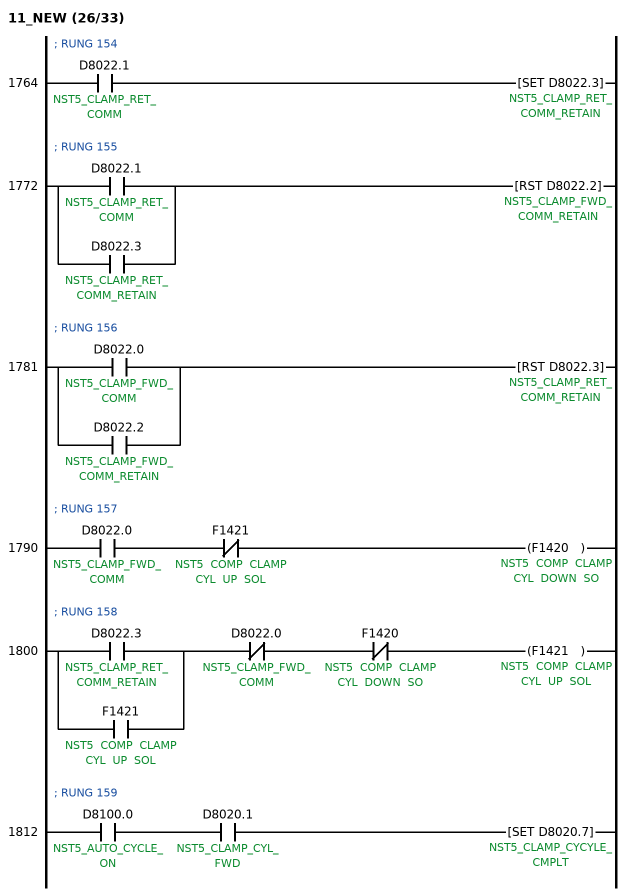
[picture p216: ladder of 11_NEW, rungs at steps 1764 to 1812]
; RUNG 154
1764  LD      D8022.1  ; NST5_CLAMP_RET_COMM
      SET     D8022.3  ; NST5_CLAMP_RET_COMM_RETAIN
; RUNG 155
1772  LD      D8022.1  ; NST5_CLAMP_RET_COMM
      OR      D8022.3  ; NST5_CLAMP_RET_COMM_RETAIN
      RST     D8022.2  ; NST5_CLAMP_FWD_COMM_RETAIN
; RUNG 156
1781  LD      D8022.0  ; NST5_CLAMP_FWD_COMM
      OR      D8022.2  ; NST5_CLAMP_FWD_COMM_RETAIN
      RST     D8022.3  ; NST5_CLAMP_RET_COMM_RETAIN
; RUNG 157
1790  LD      D8022.0  ; NST5_CLAMP_FWD_COMM
      ANI     F1421  ; NST5  COMP  CLAMP  CYL  UP  SOL
      OUT     F1420  ; NST5  COMP  CLAMP  CYL  DOWN  SO
; RUNG 158
1800  LD      D8022.3  ; NST5_CLAMP_RET_COMM_RETAIN
      OR      F1421  ; NST5  COMP  CLAMP  CYL  UP  SOL
      ANI     D8022.0  ; NST5_CLAMP_FWD_COMM
      ANI     F1420  ; NST5  COMP  CLAMP  CYL  DOWN  SO
      OUT     F1421  ; NST5  COMP  CLAMP  CYL  UP  SOL
; RUNG 159
1812  LD      D8100.0  ; NST5_AUTO_CYCLE_ON
      AND     D8020.1  ; NST5_CLAMP_CYL_FWD
      SET     D8020.7  ; NST5_CLAMP_CYCYLE_CMPLT
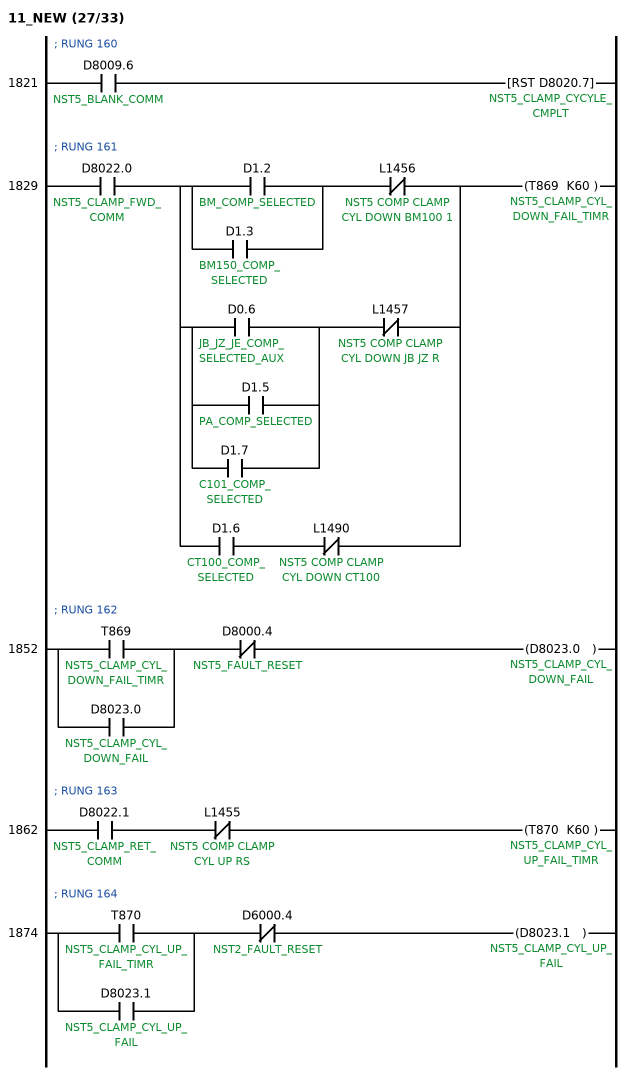
; RUNG 160
1821  LD      D8009.6  ; NST5_BLANK_COMM
      RST     D8020.7  ; NST5_CLAMP_CYCYLE_CMPLT
; RUNG 161
1829  LD      D8022.0  ; NST5_CLAMP_FWD_COMM
      LD      D1.2  ; BM_COMP_SELECTED
      OR      D1.3  ; BM150_COMP_SELECTED
      ANI     L1456  ; NST5 COMP CLAMP CYL DOWN BM100 1
      LD      D0.6  ; JB_JZ_JE_COMP_SELECTED_AUX
      OR      D1.5  ; PA_COMP_SELECTED
      OR      D1.7  ; C101_COMP_SELECTED
      ANI     L1457  ; NST5 COMP CLAMP CYL DOWN JB JZ R
      ORB
      LD      D1.6  ; CT100_COMP_SELECTED
      ANI     L1490  ; NST5 COMP CLAMP CYL DOWN CT100
      ORB
      ANB
      OUT     T869 K60  ; NST5_CLAMP_CYL_DOWN_FAIL_TIMR
; RUNG 162
1852  LD      T869  ; NST5_CLAMP_CYL_DOWN_FAIL_TIMR
      OR      D8023.0  ; NST5_CLAMP_CYL_DOWN_FAIL
      ANI     D8000.4  ; NST5_FAULT_RESET
      OUT     D8023.0  ; NST5_CLAMP_CYL_DOWN_FAIL
; RUNG 163
1862  LD      D8022.1  ; NST5_CLAMP_RET_COMM
      ANI     L1455  ; NST5 COMP CLAMP CYL UP RS
      OUT     T870 K60  ; NST5_CLAMP_CYL_UP_FAIL_TIMR
; RUNG 164
1874  LD      T870  ; NST5_CLAMP_CYL_UP_FAIL_TIMR
      OR      D8023.1  ; NST5_CLAMP_CYL_UP_FAIL
      ANI     D6000.4  ; NST2_FAULT_RESET
      OUT     D8023.1  ; NST5_CLAMP_CYL_UP_FAIL
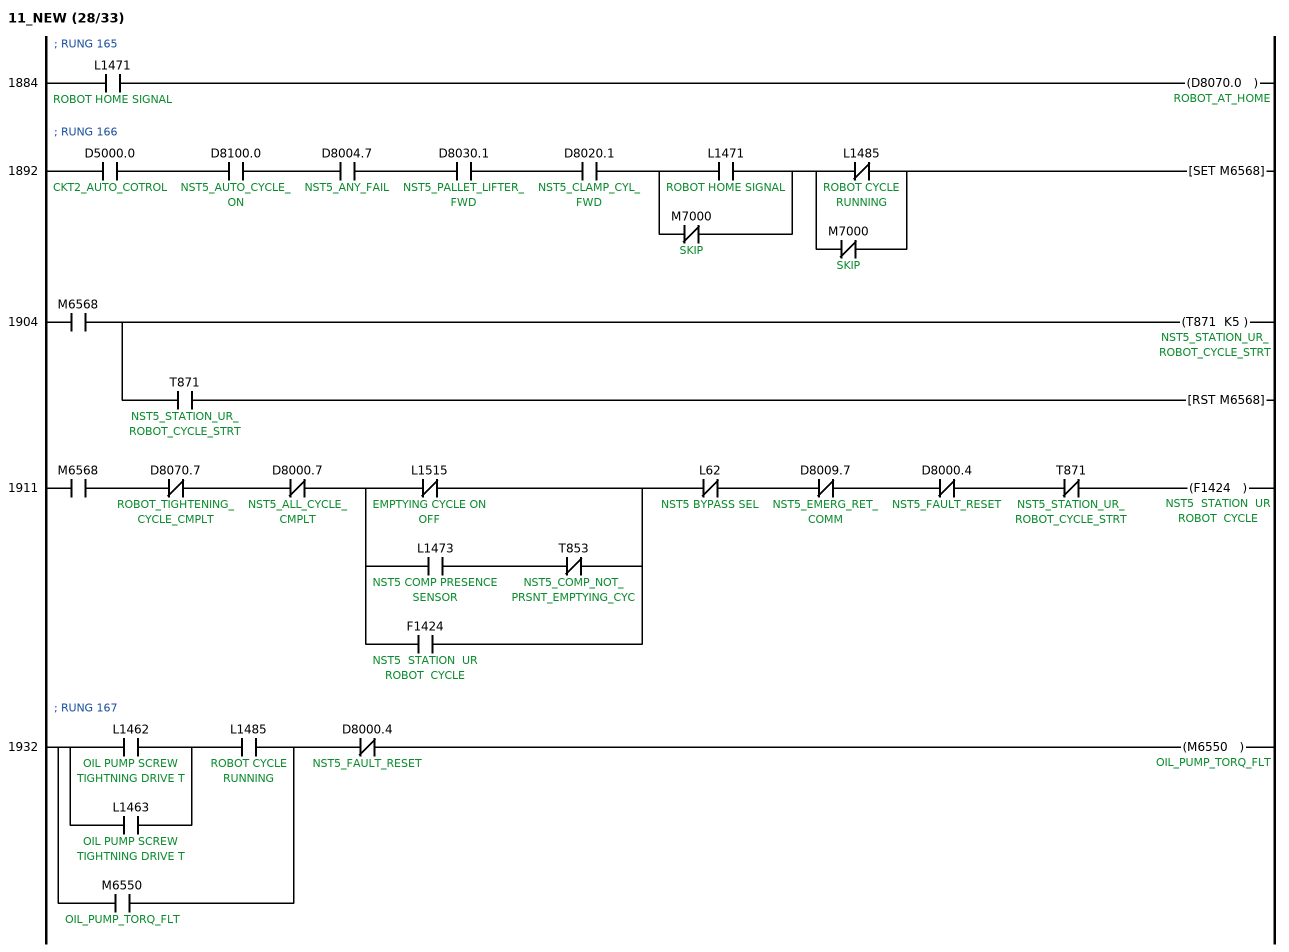
; RUNG 165
1884  LD      L1471  ; ROBOT HOME SIGNAL
      OUT     D8070.0  ; ROBOT_AT_HOME
; RUNG 166
1892  LD      D5000.0  ; CKT2_AUTO_COTROL
      AND     D8100.0  ; NST5_AUTO_CYCLE_ON
      AND     D8004.7  ; NST5_ANY_FAIL
      AND     D8030.1  ; NST5_PALLET_LIFTER_FWD
      AND     D8020.1  ; NST5_CLAMP_CYL_FWD
      LD      L1471  ; ROBOT HOME SIGNAL
      ORI     M7000  ; SKIP
      ANB
      LDI     L1485  ; ROBOT CYCLE RUNNING
      ORI     M7000  ; SKIP
      ANB
      SET     M6568
1904  LD      M6568
      OUT     T871 K5  ; NST5_STATION_UR_ROBOT_CYCLE_STRT
      AND     T871  ; NST5_STATION_UR_ROBOT_CYCLE_STRT
      RST     M6568
1911  LD      M6568
      ANI     D8070.7  ; ROBOT_TIGHTENING_CYCLE_CMPLT
      ANI     D8000.7  ; NST5_ALL_CYCLE_CMPLT
      LDI     L1515  ; EMPTYING CYCLE ON OFF
      LD      L1473  ; NST5 COMP PRESENCE SENSOR
      ANI     T853  ; NST5_COMP_NOT_PRSNT_EMPTYING_CYC
      ORB
      OR      F1424  ; NST5  STATION  UR  ROBOT  CYCLE
      ANB
      ANI     L62  ; NST5 BYPASS SEL
      ANI     D8009.7  ; NST5_EMERG_RET_COMM
      ANI     D8000.4  ; NST5_FAULT_RESET
      ANI     T871  ; NST5_STATION_UR_ROBOT_CYCLE_STRT
      OUT     F1424  ; NST5  STATION  UR  ROBOT  CYCLE
; RUNG 167
1932  LD      L1462  ; OIL PUMP SCREW TIGHTNING DRIVE T
      OR      L1463  ; OIL PUMP SCREW TIGHTNING DRIVE T
      AND     L1485  ; ROBOT CYCLE RUNNING
      OR      M6550  ; OIL_PUMP_TORQ_FLT
      ANI     D8000.4  ; NST5_FAULT_RESET
      OUT     M6550  ; OIL_PUMP_TORQ_FLT
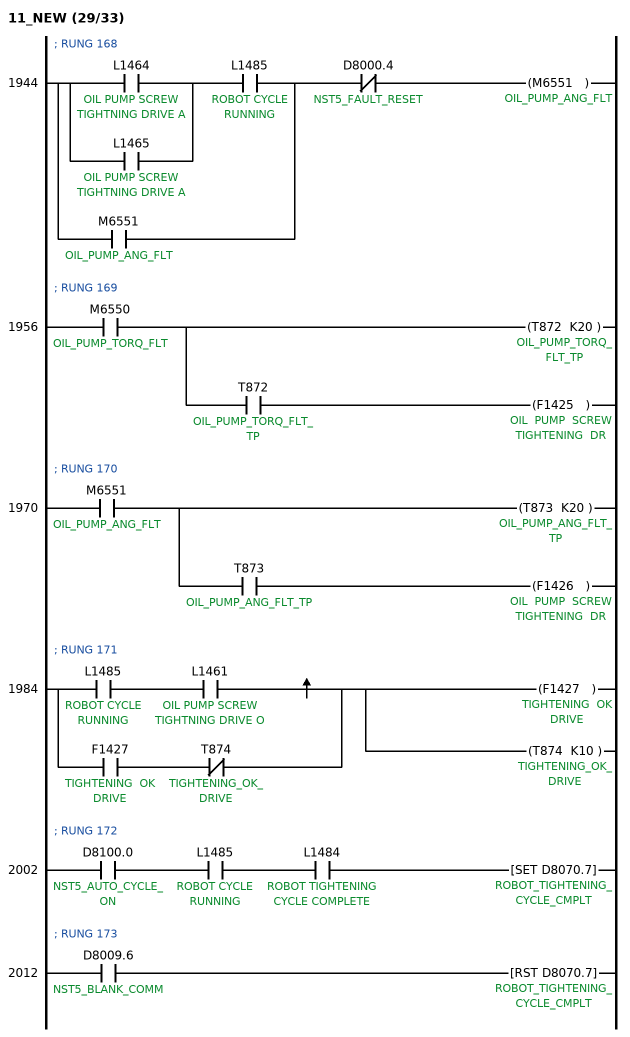
; RUNG 168
1944  LD      L1464  ; OIL PUMP SCREW TIGHTNING DRIVE A
      OR      L1465  ; OIL PUMP SCREW TIGHTNING DRIVE A
      AND     L1485  ; ROBOT CYCLE RUNNING
      OR      M6551  ; OIL_PUMP_ANG_FLT
      ANI     D8000.4  ; NST5_FAULT_RESET
      OUT     M6551  ; OIL_PUMP_ANG_FLT
; RUNG 169
1956  LD      M6550  ; OIL_PUMP_TORQ_FLT
      OUT     T872 K20  ; OIL_PUMP_TORQ_FLT_TP
      AND     T872  ; OIL_PUMP_TORQ_FLT_TP
      OUT     F1425  ; OIL  PUMP  SCREW  TIGHTENING  DR
; RUNG 170
1970  LD      M6551  ; OIL_PUMP_ANG_FLT
      OUT     T873 K20  ; OIL_PUMP_ANG_FLT_TP
      AND     T873  ; OIL_PUMP_ANG_FLT_TP
      OUT     F1426  ; OIL  PUMP  SCREW  TIGHTENING  DR
; RUNG 171
1984  LD      L1485  ; ROBOT CYCLE RUNNING
      AND     L1461  ; OIL PUMP SCREW TIGHTNING DRIVE O
      MEP
      LD      F1427  ; TIGHTENING  OK  DRIVE
      ANI     T874  ; TIGHTENING_OK_DRIVE
      ORB
      OUT     F1427  ; TIGHTENING  OK  DRIVE
      OUT     T874 K10  ; TIGHTENING_OK_DRIVE
; RUNG 172
2002  LD      D8100.0  ; NST5_AUTO_CYCLE_ON
      AND     L1485  ; ROBOT CYCLE RUNNING
      AND     L1484  ; ROBOT TIGHTENING CYCLE COMPLETE
      SET     D8070.7  ; ROBOT_TIGHTENING_CYCLE_CMPLT
; RUNG 173
2012  LD      D8009.6  ; NST5_BLANK_COMM
      RST     D8070.7  ; ROBOT_TIGHTENING_CYCLE_CMPLT
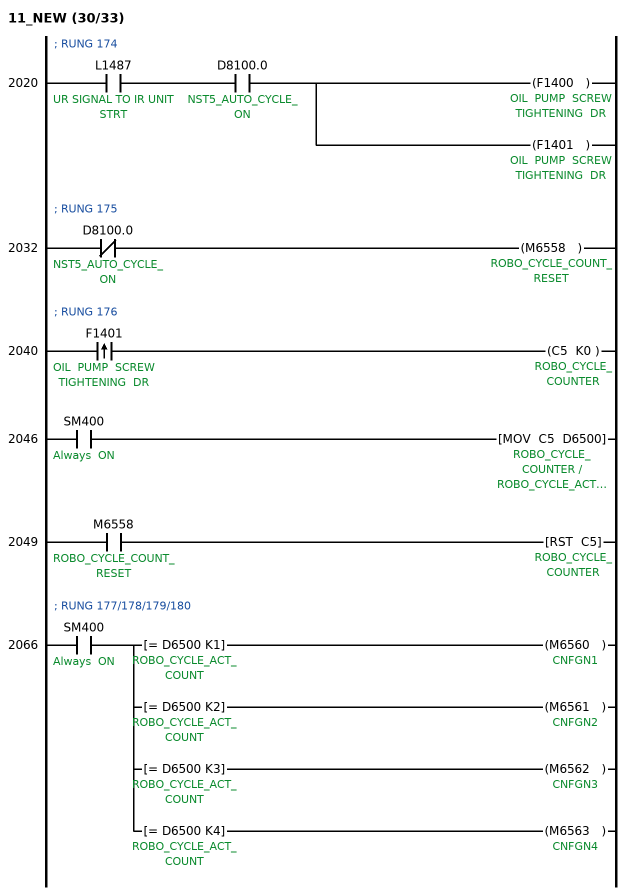
; RUNG 174
2020  LD      L1487  ; UR SIGNAL TO IR UNIT STRT
      AND     D8100.0  ; NST5_AUTO_CYCLE_ON
      OUT     F1400  ; OIL  PUMP  SCREW  TIGHTENING  DR
      OUT     F1401  ; OIL  PUMP  SCREW  TIGHTENING  DR
; RUNG 175
2032  LDI     D8100.0  ; NST5_AUTO_CYCLE_ON
      OUT     M6558  ; ROBO_CYCLE_COUNT_RESET
; RUNG 176
2040  LDP     F1401  ; OIL  PUMP  SCREW  TIGHTENING  DR
      OUT     C5 K0  ; ROBO_CYCLE_COUNTER
2046  LD      SM400  ; Always  ON
      MOV     C5 D6500  ; ROBO_CYCLE_ACT_COUNT
2049  LD      M6558  ; ROBO_CYCLE_COUNT_RESET
      RST     C5  ; ROBO_CYCLE_COUNTER
; RUNG 177/178/179/180
2066  LD      SM400  ; Always  ON
      MPS
      AND=    D6500 K1  ; ROBO_CYCLE_ACT_COUNT
      OUT     M6560  ; CNFGN1
      MRD
      AND=    D6500 K2  ; ROBO_CYCLE_ACT_COUNT
      OUT     M6561  ; CNFGN2
      MRD
      AND=    D6500 K3  ; ROBO_CYCLE_ACT_COUNT
      OUT     M6562  ; CNFGN3
      MPP
      AND=    D6500 K4  ; ROBO_CYCLE_ACT_COUNT
      OUT     M6563  ; CNFGN4
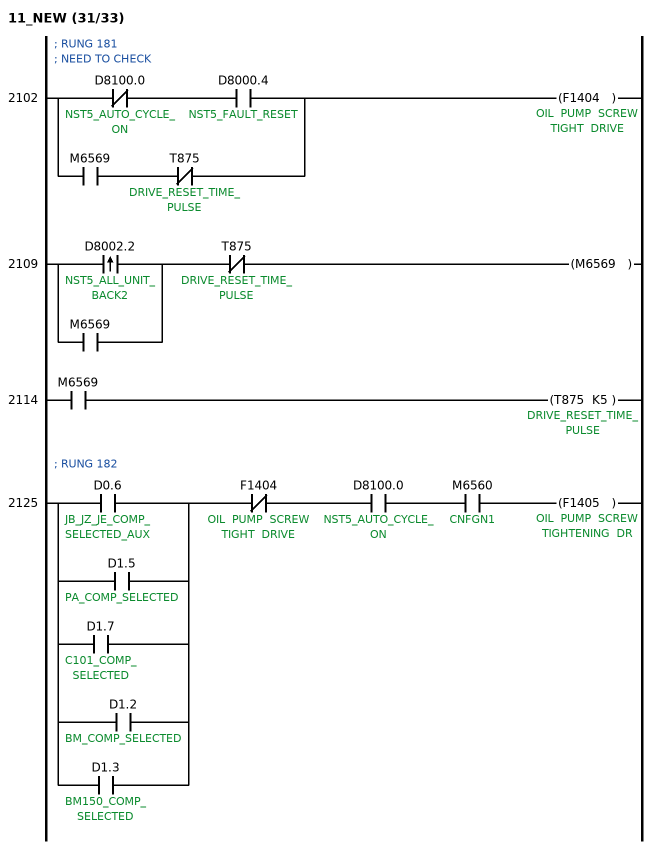
; RUNG 181
; NEED TO CHECK
2102  LDI     D8100.0  ; NST5_AUTO_CYCLE_ON
      AND     D8000.4  ; NST5_FAULT_RESET
      LD      M6569
      ANI     T875  ; DRIVE_RESET_TIME_PULSE
      ORB
      OUT     F1404  ; OIL  PUMP  SCREW  TIGHT  DRIVE
2109  LDP     D8002.2  ; NST5_ALL_UNIT_BACK2
      OR      M6569
      ANI     T875  ; DRIVE_RESET_TIME_PULSE
      OUT     M6569
2114  LD      M6569
      OUT     T875 K5  ; DRIVE_RESET_TIME_PULSE
; RUNG 182
2125  LD      D0.6  ; JB_JZ_JE_COMP_SELECTED_AUX
      OR      D1.5  ; PA_COMP_SELECTED
      OR      D1.7  ; C101_COMP_SELECTED
      OR      D1.2  ; BM_COMP_SELECTED
      OR      D1.3  ; BM150_COMP_SELECTED
      ANI     F1404  ; OIL  PUMP  SCREW  TIGHT  DRIVE
      AND     D8100.0  ; NST5_AUTO_CYCLE_ON
      AND     M6560  ; CNFGN1
      OUT     F1405  ; OIL  PUMP  SCREW  TIGHTENING  DR
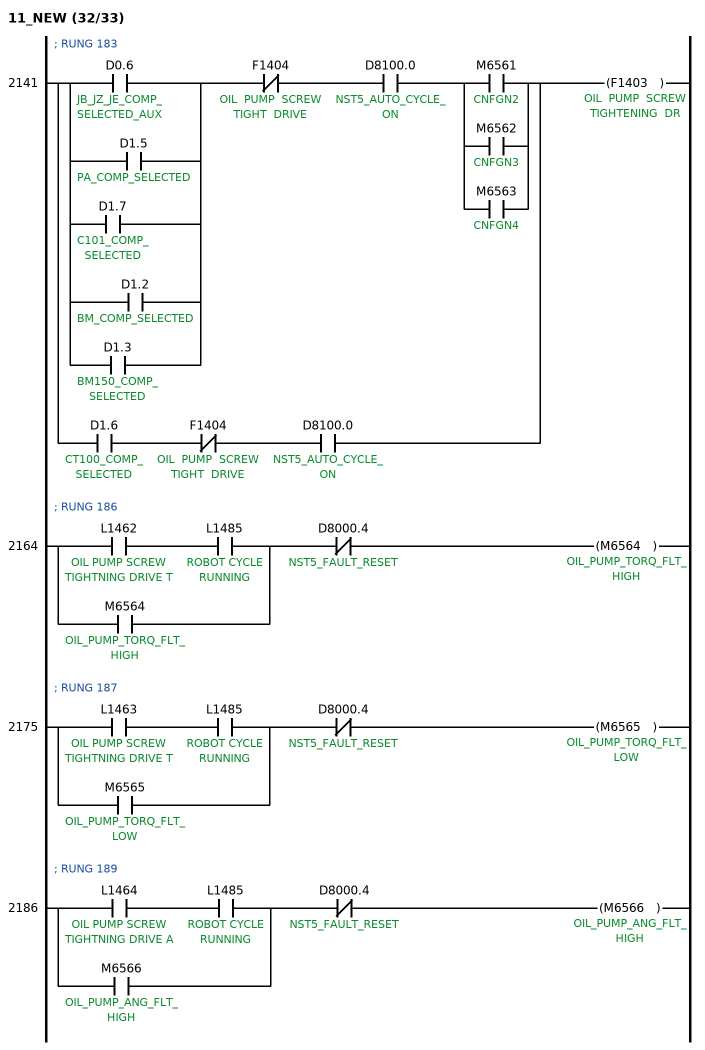
; RUNG 183
2141  LD      D0.6  ; JB_JZ_JE_COMP_SELECTED_AUX
      OR      D1.5  ; PA_COMP_SELECTED
      OR      D1.7  ; C101_COMP_SELECTED
      OR      D1.2  ; BM_COMP_SELECTED
      OR      D1.3  ; BM150_COMP_SELECTED
      ANI     F1404  ; OIL  PUMP  SCREW  TIGHT  DRIVE
      AND     D8100.0  ; NST5_AUTO_CYCLE_ON
      LD      M6561  ; CNFGN2
      OR      M6562  ; CNFGN3
      OR      M6563  ; CNFGN4
      ANB
      LD      D1.6  ; CT100_COMP_SELECTED
      ANI     F1404  ; OIL  PUMP  SCREW  TIGHT  DRIVE
      AND     D8100.0  ; NST5_AUTO_CYCLE_ON
      ORB
      OUT     F1403  ; OIL  PUMP  SCREW  TIGHTENING  DR
; RUNG 186
2164  LD      L1462  ; OIL PUMP SCREW TIGHTNING DRIVE T
      AND     L1485  ; ROBOT CYCLE RUNNING
      OR      M6564  ; OIL_PUMP_TORQ_FLT_HIGH
      ANI     D8000.4  ; NST5_FAULT_RESET
      OUT     M6564  ; OIL_PUMP_TORQ_FLT_HIGH
; RUNG 187
2175  LD      L1463  ; OIL PUMP SCREW TIGHTNING DRIVE T
      AND     L1485  ; ROBOT CYCLE RUNNING
      OR      M6565  ; OIL_PUMP_TORQ_FLT_LOW
      ANI     D8000.4  ; NST5_FAULT_RESET
      OUT     M6565  ; OIL_PUMP_TORQ_FLT_LOW
; RUNG 189
2186  LD      L1464  ; OIL PUMP SCREW TIGHTNING DRIVE A
      AND     L1485  ; ROBOT CYCLE RUNNING
      OR      M6566  ; OIL_PUMP_ANG_FLT_HIGH
      ANI     D8000.4  ; NST5_FAULT_RESET
      OUT     M6566  ; OIL_PUMP_ANG_FLT_HIGH
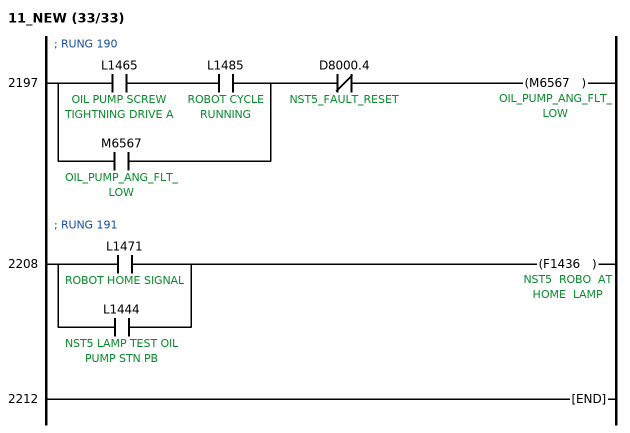
; RUNG 190
2197  LD      L1465  ; OIL PUMP SCREW TIGHTNING DRIVE A
      AND     L1485  ; ROBOT CYCLE RUNNING
      OR      M6567  ; OIL_PUMP_ANG_FLT_LOW
      ANI     D8000.4  ; NST5_FAULT_RESET
      OUT     M6567  ; OIL_PUMP_ANG_FLT_LOW
; RUNG 191
2208  LD      L1471  ; ROBOT HOME SIGNAL
      OR      L1444  ; NST5 LAMP TEST OIL PUMP STN PB
      OUT     F1436  ; NST5  ROBO  AT  HOME  LAMP
2212  END
END_PROGRAM

PROGRAM 12_NEW  // ST5 CK2 AUX
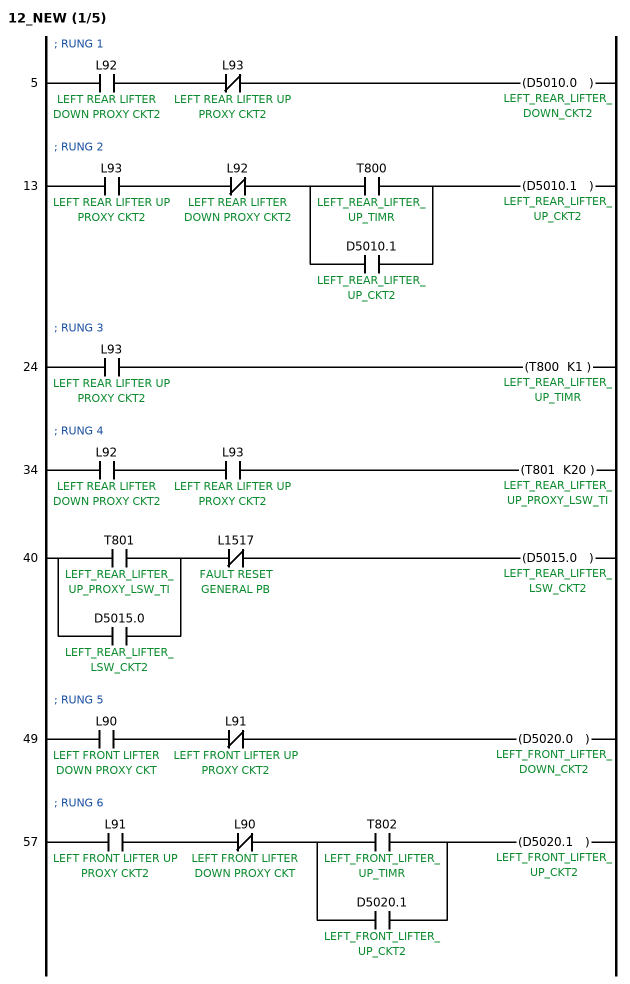
; RUNG 1
5     LD      L92  ; LEFT REAR LIFTER DOWN PROXY CKT2
      ANI     L93  ; LEFT REAR LIFTER UP PROXY CKT2
      OUT     D5010.0  ; LEFT_REAR_LIFTER_DOWN_CKT2
; RUNG 2
13    LD      L93  ; LEFT REAR LIFTER UP PROXY CKT2
      ANI     L92  ; LEFT REAR LIFTER DOWN PROXY CKT2
      LD      T800  ; LEFT_REAR_LIFTER_UP_TIMR
      OR      D5010.1  ; LEFT_REAR_LIFTER_UP_CKT2
      ANB
      OUT     D5010.1  ; LEFT_REAR_LIFTER_UP_CKT2
; RUNG 3
24    LD      L93  ; LEFT REAR LIFTER UP PROXY CKT2
      OUT     T800 K1  ; LEFT_REAR_LIFTER_UP_TIMR
; RUNG 4
34    LD      L92  ; LEFT REAR LIFTER DOWN PROXY CKT2
      AND     L93  ; LEFT REAR LIFTER UP PROXY CKT2
      OUT     T801 K20  ; LEFT_REAR_LIFTER_UP_PROXY_LSW_TI
40    LD      T801  ; LEFT_REAR_LIFTER_UP_PROXY_LSW_TI
      OR      D5015.0  ; LEFT_REAR_LIFTER_LSW_CKT2
      ANI     L1517  ; FAULT RESET GENERAL PB
      OUT     D5015.0  ; LEFT_REAR_LIFTER_LSW_CKT2
; RUNG 5
49    LD      L90  ; LEFT FRONT LIFTER DOWN PROXY CKT
      ANI     L91  ; LEFT FRONT LIFTER UP PROXY CKT2
      OUT     D5020.0  ; LEFT_FRONT_LIFTER_DOWN_CKT2
; RUNG 6
57    LD      L91  ; LEFT FRONT LIFTER UP PROXY CKT2
      ANI     L90  ; LEFT FRONT LIFTER DOWN PROXY CKT
      LD      T802  ; LEFT_FRONT_LIFTER_UP_TIMR
      OR      D5020.1  ; LEFT_FRONT_LIFTER_UP_CKT2
      ANB
      OUT     D5020.1  ; LEFT_FRONT_LIFTER_UP_CKT2
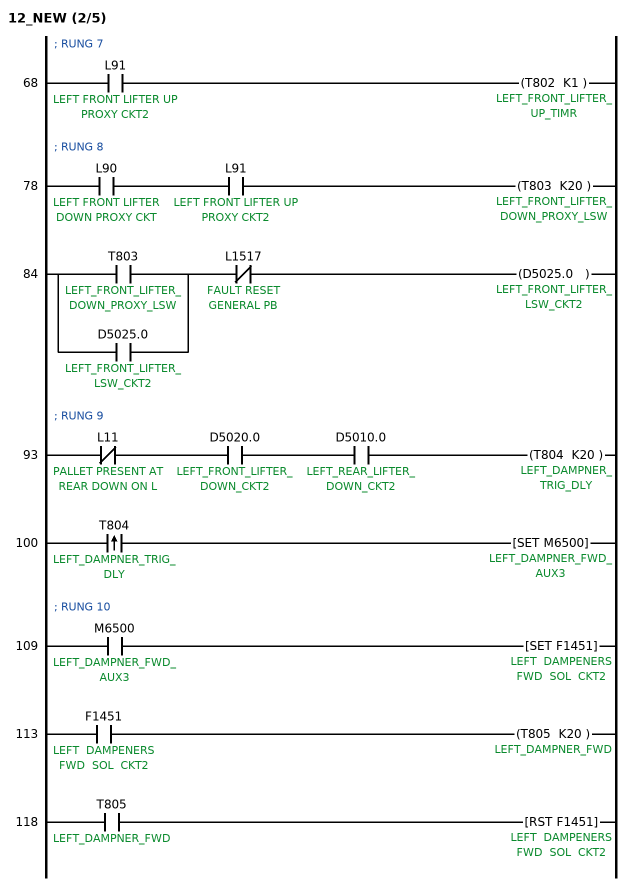
; RUNG 7
68    LD      L91  ; LEFT FRONT LIFTER UP PROXY CKT2
      OUT     T802 K1  ; LEFT_FRONT_LIFTER_UP_TIMR
; RUNG 8
78    LD      L90  ; LEFT FRONT LIFTER DOWN PROXY CKT
      AND     L91  ; LEFT FRONT LIFTER UP PROXY CKT2
      OUT     T803 K20  ; LEFT_FRONT_LIFTER_DOWN_PROXY_LSW
84    LD      T803  ; LEFT_FRONT_LIFTER_DOWN_PROXY_LSW
      OR      D5025.0  ; LEFT_FRONT_LIFTER_LSW_CKT2
      ANI     L1517  ; FAULT RESET GENERAL PB
      OUT     D5025.0  ; LEFT_FRONT_LIFTER_LSW_CKT2
; RUNG 9
93    LDI     L11  ; PALLET PRESENT AT REAR DOWN ON L
      AND     D5020.0  ; LEFT_FRONT_LIFTER_DOWN_CKT2
      AND     D5010.0  ; LEFT_REAR_LIFTER_DOWN_CKT2
      OUT     T804 K20  ; LEFT_DAMPNER_TRIG_DLY
100   LDP     T804  ; LEFT_DAMPNER_TRIG_DLY
      SET     M6500  ; LEFT_DAMPNER_FWD_AUX3
; RUNG 10
109   LD      M6500  ; LEFT_DAMPNER_FWD_AUX3
      SET     F1451  ; LEFT  DAMPENERS  FWD  SOL  CKT2
113   LD      F1451  ; LEFT  DAMPENERS  FWD  SOL  CKT2
      OUT     T805 K20  ; LEFT_DAMPNER_FWD
118   LD      T805  ; LEFT_DAMPNER_FWD
      RST     F1451  ; LEFT  DAMPENERS  FWD  SOL  CKT2
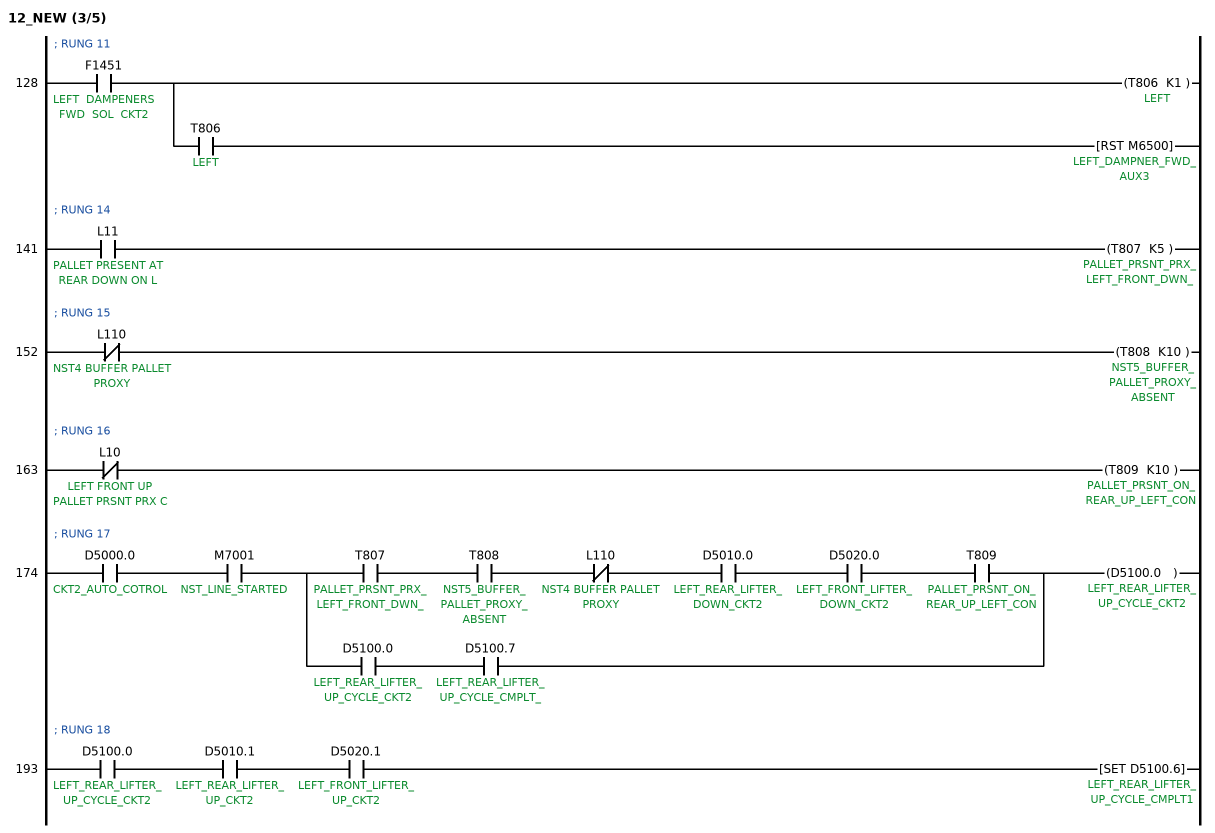
; RUNG 11
128   LD      F1451  ; LEFT  DAMPENERS  FWD  SOL  CKT2
      OUT     T806 K1  ; LEFT
      AND     T806  ; LEFT
      RST     M6500  ; LEFT_DAMPNER_FWD_AUX3
; RUNG 14
141   LD      L11  ; PALLET PRESENT AT REAR DOWN ON L
      OUT     T807 K5  ; PALLET_PRSNT_PRX_LEFT_FRONT_DWN_
; RUNG 15
152   LDI     L110  ; NST4 BUFFER PALLET PROXY
      OUT     T808 K10  ; NST5_BUFFER_PALLET_PROXY_ABSENT
; RUNG 16
163   LDI     L10  ; LEFT FRONT UP PALLET PRSNT PRX C
      OUT     T809 K10  ; PALLET_PRSNT_ON_REAR_UP_LEFT_CON
; RUNG 17
174   LD      D5000.0  ; CKT2_AUTO_COTROL
      AND     M7001  ; NST_LINE_STARTED
      LD      T807  ; PALLET_PRSNT_PRX_LEFT_FRONT_DWN_
      AND     T808  ; NST5_BUFFER_PALLET_PROXY_ABSENT
      ANI     L110  ; NST4 BUFFER PALLET PROXY
      AND     D5010.0  ; LEFT_REAR_LIFTER_DOWN_CKT2
      AND     D5020.0  ; LEFT_FRONT_LIFTER_DOWN_CKT2
      AND     T809  ; PALLET_PRSNT_ON_REAR_UP_LEFT_CON
      LD      D5100.0  ; LEFT_REAR_LIFTER_UP_CYCLE_CKT2
      AND     D5100.7  ; LEFT_REAR_LIFTER_UP_CYCLE_CMPLT_
      ORB
      ANB
      OUT     D5100.0  ; LEFT_REAR_LIFTER_UP_CYCLE_CKT2
; RUNG 18
193   LD      D5100.0  ; LEFT_REAR_LIFTER_UP_CYCLE_CKT2
      AND     D5010.1  ; LEFT_REAR_LIFTER_UP_CKT2
      AND     D5020.1  ; LEFT_FRONT_LIFTER_UP_CKT2
      SET     D5100.6  ; LEFT_REAR_LIFTER_UP_CYCLE_CMPLT1
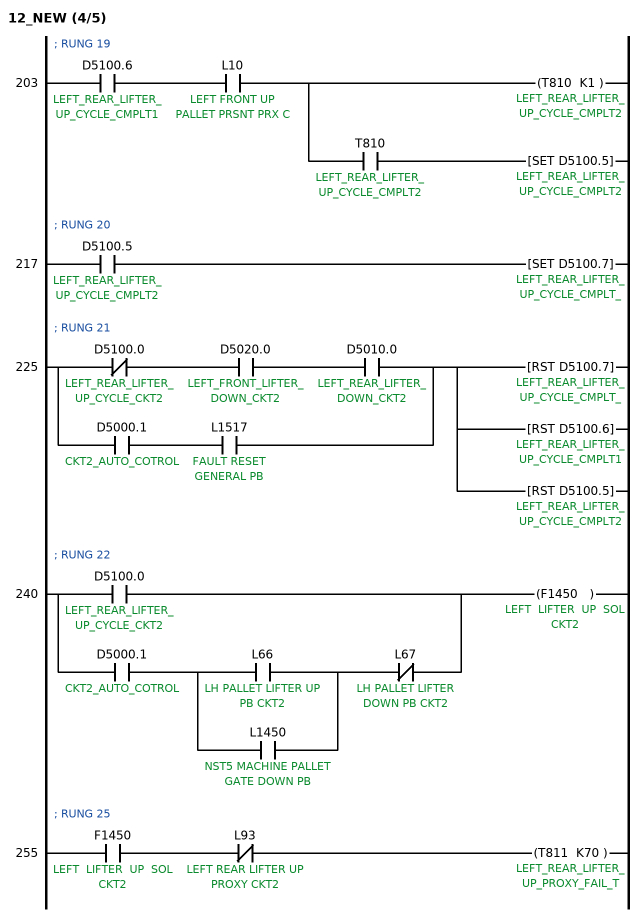
; RUNG 19
203   LD      D5100.6  ; LEFT_REAR_LIFTER_UP_CYCLE_CMPLT1
      AND     L10  ; LEFT FRONT UP PALLET PRSNT PRX C
      OUT     T810 K1  ; LEFT_REAR_LIFTER_UP_CYCLE_CMPLT2
      AND     T810  ; LEFT_REAR_LIFTER_UP_CYCLE_CMPLT2
      SET     D5100.5  ; LEFT_REAR_LIFTER_UP_CYCLE_CMPLT2
; RUNG 20
217   LD      D5100.5  ; LEFT_REAR_LIFTER_UP_CYCLE_CMPLT2
      SET     D5100.7  ; LEFT_REAR_LIFTER_UP_CYCLE_CMPLT_
; RUNG 21
225   LDI     D5100.0  ; LEFT_REAR_LIFTER_UP_CYCLE_CKT2
      AND     D5020.0  ; LEFT_FRONT_LIFTER_DOWN_CKT2
      AND     D5010.0  ; LEFT_REAR_LIFTER_DOWN_CKT2
      LD      D5000.1  ; CKT2_AUTO_COTROL
      AND     L1517  ; FAULT RESET GENERAL PB
      ORB
      RST     D5100.7  ; LEFT_REAR_LIFTER_UP_CYCLE_CMPLT_
      RST     D5100.6  ; LEFT_REAR_LIFTER_UP_CYCLE_CMPLT1
      RST     D5100.5  ; LEFT_REAR_LIFTER_UP_CYCLE_CMPLT2
; RUNG 22
240   LD      D5100.0  ; LEFT_REAR_LIFTER_UP_CYCLE_CKT2
      LD      D5000.1  ; CKT2_AUTO_COTROL
      LD      L66  ; LH PALLET LIFTER UP PB CKT2
      OR      L1450  ; NST5 MACHINE PALLET GATE DOWN PB
      ANB
      ANI     L67  ; LH PALLET LIFTER DOWN PB CKT2
      ORB
      OUT     F1450  ; LEFT  LIFTER  UP  SOL  CKT2
; RUNG 25
255   LD      F1450  ; LEFT  LIFTER  UP  SOL  CKT2
      ANI     L93  ; LEFT REAR LIFTER UP PROXY CKT2
      OUT     T811 K70  ; LEFT_REAR_LIFTER_UP_PROXY_FAIL_T
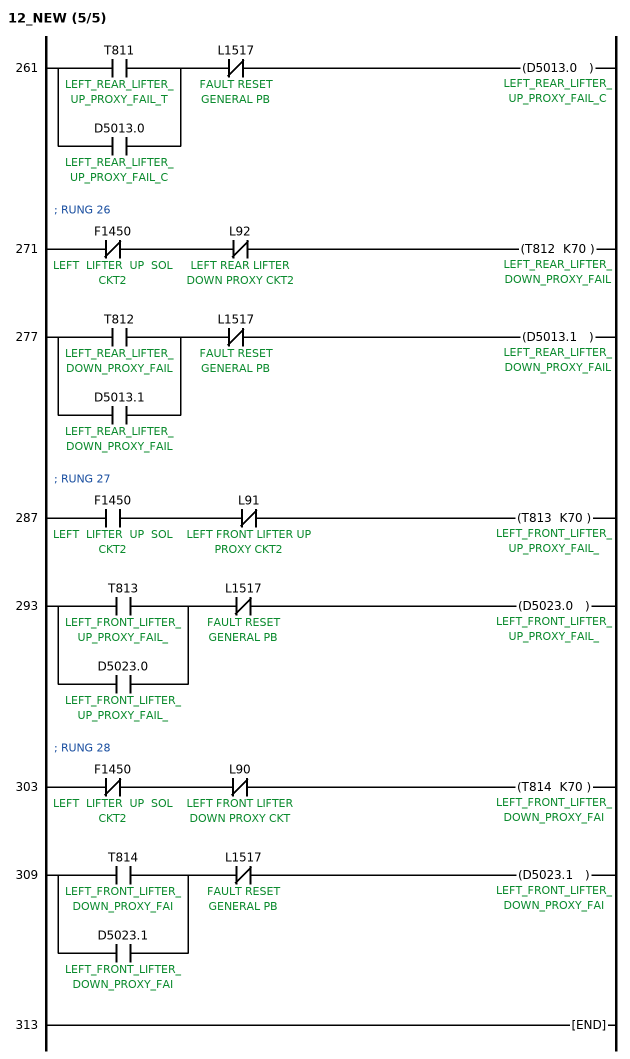
261   LD      T811  ; LEFT_REAR_LIFTER_UP_PROXY_FAIL_T
      OR      D5013.0  ; LEFT_REAR_LIFTER_UP_PROXY_FAIL_C
      ANI     L1517  ; FAULT RESET GENERAL PB
      OUT     D5013.0  ; LEFT_REAR_LIFTER_UP_PROXY_FAIL_C
; RUNG 26
271   LDI     F1450  ; LEFT  LIFTER  UP  SOL  CKT2
      ANI     L92  ; LEFT REAR LIFTER DOWN PROXY CKT2
      OUT     T812 K70  ; LEFT_REAR_LIFTER_DOWN_PROXY_FAIL
277   LD      T812  ; LEFT_REAR_LIFTER_DOWN_PROXY_FAIL
      OR      D5013.1  ; LEFT_REAR_LIFTER_DOWN_PROXY_FAIL
      ANI     L1517  ; FAULT RESET GENERAL PB
      OUT     D5013.1  ; LEFT_REAR_LIFTER_DOWN_PROXY_FAIL
; RUNG 27
287   LD      F1450  ; LEFT  LIFTER  UP  SOL  CKT2
      ANI     L91  ; LEFT FRONT LIFTER UP PROXY CKT2
      OUT     T813 K70  ; LEFT_FRONT_LIFTER_UP_PROXY_FAIL_
293   LD      T813  ; LEFT_FRONT_LIFTER_UP_PROXY_FAIL_
      OR      D5023.0  ; LEFT_FRONT_LIFTER_UP_PROXY_FAIL_
      ANI     L1517  ; FAULT RESET GENERAL PB
      OUT     D5023.0  ; LEFT_FRONT_LIFTER_UP_PROXY_FAIL_
; RUNG 28
303   LDI     F1450  ; LEFT  LIFTER  UP  SOL  CKT2
      ANI     L90  ; LEFT FRONT LIFTER DOWN PROXY CKT
      OUT     T814 K70  ; LEFT_FRONT_LIFTER_DOWN_PROXY_FAI
309   LD      T814  ; LEFT_FRONT_LIFTER_DOWN_PROXY_FAI
      OR      D5023.1  ; LEFT_FRONT_LIFTER_DOWN_PROXY_FAI
      ANI     L1517  ; FAULT RESET GENERAL PB
      OUT     D5023.1  ; LEFT_FRONT_LIFTER_DOWN_PROXY_FAI
313   END
END_PROGRAM

PROGRAM 13_NEW  // ST6 CK2
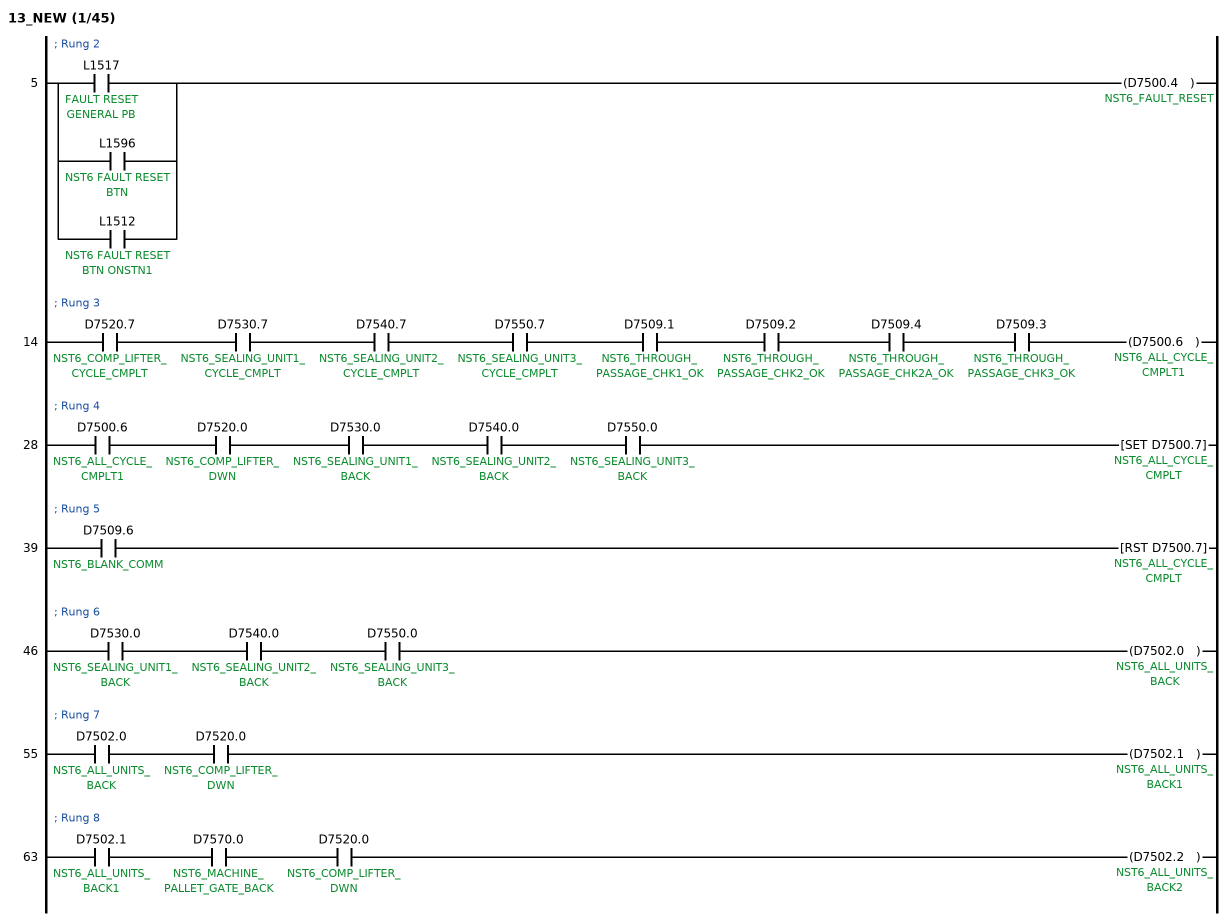
; Rung 2
5     LD      L1517  ; FAULT RESET GENERAL PB
      OR      L1596  ; NST6 FAULT RESET BTN
      OR      L1512  ; NST6 FAULT RESET BTN ONSTN1
      OUT     D7500.4  ; NST6_FAULT_RESET
; Rung 3
14    LD      D7520.7  ; NST6_COMP_LIFTER_CYCLE_CMPLT
      AND     D7530.7  ; NST6_SEALING_UNIT1_CYCLE_CMPLT
      AND     D7540.7  ; NST6_SEALING_UNIT2_CYCLE_CMPLT
      AND     D7550.7  ; NST6_SEALING_UNIT3_CYCLE_CMPLT
      AND     D7509.1  ; NST6_THROUGH_PASSAGE_CHK1_OK
      AND     D7509.2  ; NST6_THROUGH_PASSAGE_CHK2_OK
      AND     D7509.4  ; NST6_THROUGH_PASSAGE_CHK2A_OK
      AND     D7509.3  ; NST6_THROUGH_PASSAGE_CHK3_OK
      OUT     D7500.6  ; NST6_ALL_CYCLE_CMPLT1
; Rung 4
28    LD      D7500.6  ; NST6_ALL_CYCLE_CMPLT1
      AND     D7520.0  ; NST6_COMP_LIFTER_DWN
      AND     D7530.0  ; NST6_SEALING_UNIT1_BACK
      AND     D7540.0  ; NST6_SEALING_UNIT2_BACK
      AND     D7550.0  ; NST6_SEALING_UNIT3_BACK
      SET     D7500.7  ; NST6_ALL_CYCLE_CMPLT
; Rung 5
39    LD      D7509.6  ; NST6_BLANK_COMM
      RST     D7500.7  ; NST6_ALL_CYCLE_CMPLT
; Rung 6
46    LD      D7530.0  ; NST6_SEALING_UNIT1_BACK
      AND     D7540.0  ; NST6_SEALING_UNIT2_BACK
      AND     D7550.0  ; NST6_SEALING_UNIT3_BACK
      OUT     D7502.0  ; NST6_ALL_UNITS_BACK
; Rung 7
55    LD      D7502.0  ; NST6_ALL_UNITS_BACK
      AND     D7520.0  ; NST6_COMP_LIFTER_DWN
      OUT     D7502.1  ; NST6_ALL_UNITS_BACK1
; Rung 8
63    LD      D7502.1  ; NST6_ALL_UNITS_BACK1
      AND     D7570.0  ; NST6_MACHINE_PALLET_GATE_BACK
      AND     D7520.0  ; NST6_COMP_LIFTER_DWN
      OUT     D7502.2  ; NST6_ALL_UNITS_BACK2
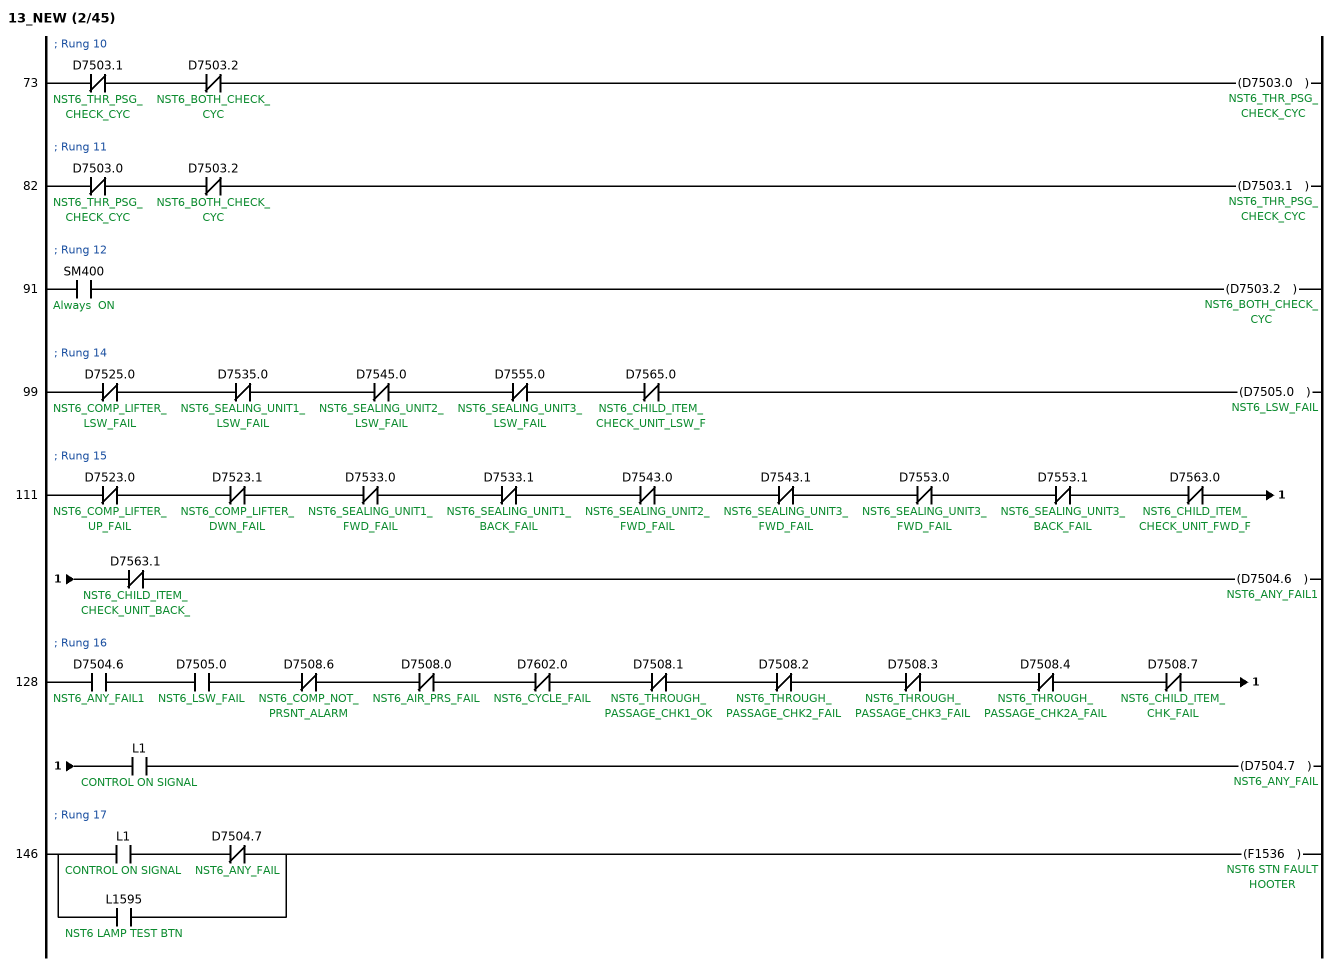
; Rung 10
73    LDI     D7503.1  ; NST6_THR_PSG_CHECK_CYC
      ANI     D7503.2  ; NST6_BOTH_CHECK_CYC
      OUT     D7503.0  ; NST6_THR_PSG_CHECK_CYC
; Rung 11
82    LDI     D7503.0  ; NST6_THR_PSG_CHECK_CYC
      ANI     D7503.2  ; NST6_BOTH_CHECK_CYC
      OUT     D7503.1  ; NST6_THR_PSG_CHECK_CYC
; Rung 12
91    LD      SM400  ; Always  ON
      OUT     D7503.2  ; NST6_BOTH_CHECK_CYC
; Rung 14
99    LDI     D7525.0  ; NST6_COMP_LIFTER_LSW_FAIL
      ANI     D7535.0  ; NST6_SEALING_UNIT1_LSW_FAIL
      ANI     D7545.0  ; NST6_SEALING_UNIT2_LSW_FAIL
      ANI     D7555.0  ; NST6_SEALING_UNIT3_LSW_FAIL
      ANI     D7565.0  ; NST6_CHILD_ITEM_CHECK_UNIT_LSW_F
      OUT     D7505.0  ; NST6_LSW_FAIL
; Rung 15
111   LDI     D7523.0  ; NST6_COMP_LIFTER_UP_FAIL
      ANI     D7523.1  ; NST6_COMP_LIFTER_DWN_FAIL
      ANI     D7533.0  ; NST6_SEALING_UNIT1_FWD_FAIL
      ANI     D7533.1  ; NST6_SEALING_UNIT1_BACK_FAIL
      ANI     D7543.0  ; NST6_SEALING_UNIT2_FWD_FAIL
      ANI     D7543.1  ; NST6_SEALING_UNIT3_FWD_FAIL
      ANI     D7553.0  ; NST6_SEALING_UNIT3_FWD_FAIL
      ANI     D7553.1  ; NST6_SEALING_UNIT3_BACK_FAIL
      ANI     D7563.0  ; NST6_CHILD_ITEM_CHECK_UNIT_FWD_F
      ANI     D7563.1  ; NST6_CHILD_ITEM_CHECK_UNIT_BACK_
      OUT     D7504.6  ; NST6_ANY_FAIL1
; Rung 16
128   LD      D7504.6  ; NST6_ANY_FAIL1
      AND     D7505.0  ; NST6_LSW_FAIL
      ANI     D7508.6  ; NST6_COMP_NOT_PRSNT_ALARM
      ANI     D7508.0  ; NST6_AIR_PRS_FAIL
      ANI     D7602.0  ; NST6_CYCLE_FAIL
      ANI     D7508.1  ; NST6_THROUGH_PASSAGE_CHK1_OK
      ANI     D7508.2  ; NST6_THROUGH_PASSAGE_CHK2_FAIL
      ANI     D7508.3  ; NST6_THROUGH_PASSAGE_CHK3_FAIL
      ANI     D7508.4  ; NST6_THROUGH_PASSAGE_CHK2A_FAIL
      ANI     D7508.7  ; NST6_CHILD_ITEM_CHK_FAIL
      AND     L1  ; CONTROL ON SIGNAL
      OUT     D7504.7  ; NST6_ANY_FAIL
; Rung 17
146   LD      L1  ; CONTROL ON SIGNAL
      ANI     D7504.7  ; NST6_ANY_FAIL
      OR      L1595  ; NST6 LAMP TEST BTN
      OUT     F1536  ; NST6 STN FAULT HOOTER
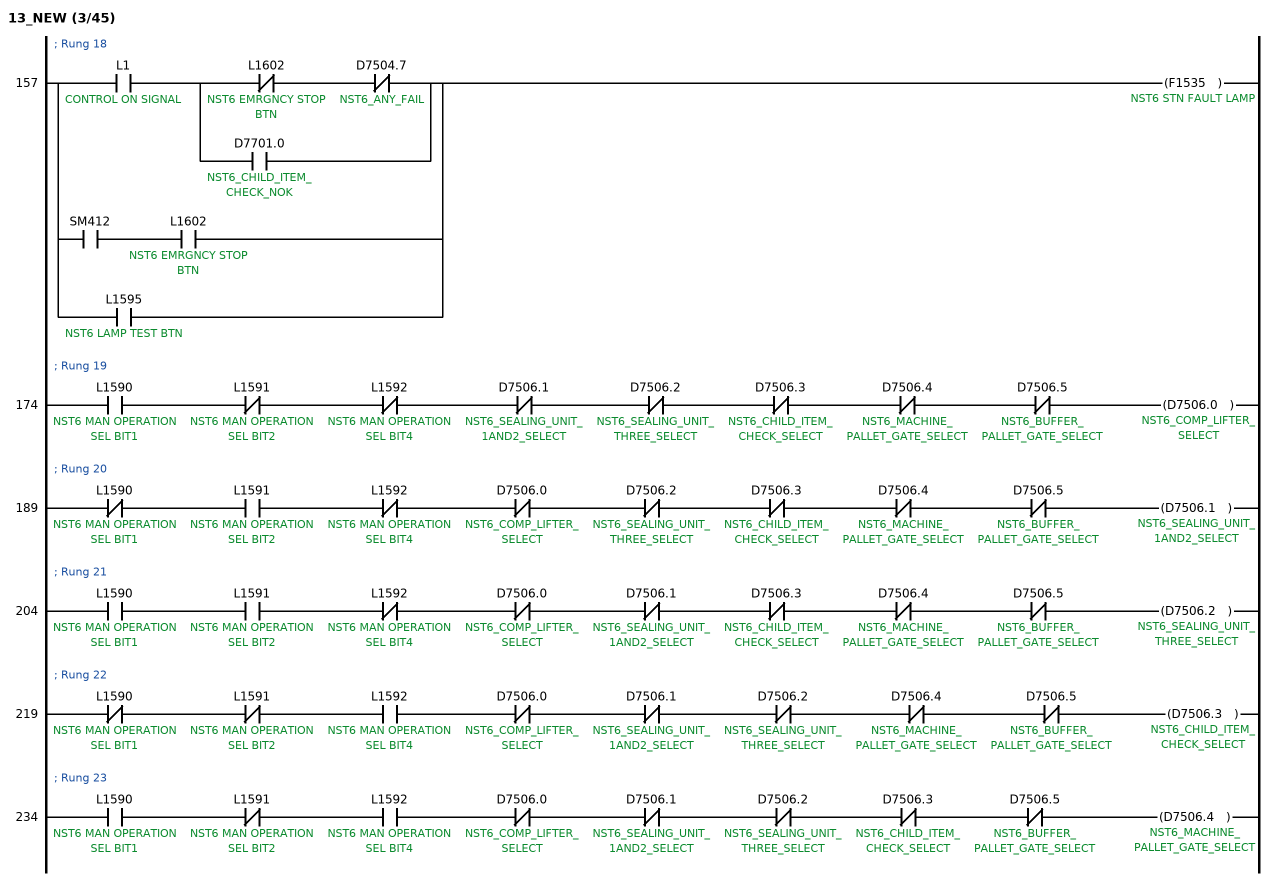
; Rung 18
157   LD      L1  ; CONTROL ON SIGNAL
      LDI     L1602  ; NST6 EMRGNCY STOP BTN
      ANI     D7504.7  ; NST6_ANY_FAIL
      OR      D7701.0  ; NST6_CHILD_ITEM_CHECK_NOK
      ANB
      LD      SM412
      AND     L1602  ; NST6 EMRGNCY STOP BTN
      ORB
      OR      L1595  ; NST6 LAMP TEST BTN
      OUT     F1535  ; NST6 STN FAULT LAMP
; Rung 19
174   LD      L1590  ; NST6 MAN OPERATION SEL BIT1
      ANI     L1591  ; NST6 MAN OPERATION SEL BIT2
      ANI     L1592  ; NST6 MAN OPERATION SEL BIT4
      ANI     D7506.1  ; NST6_SEALING_UNIT_1AND2_SELECT
      ANI     D7506.2  ; NST6_SEALING_UNIT_THREE_SELECT
      ANI     D7506.3  ; NST6_CHILD_ITEM_CHECK_SELECT
      ANI     D7506.4  ; NST6_MACHINE_PALLET_GATE_SELECT
      ANI     D7506.5  ; NST6_BUFFER_PALLET_GATE_SELECT
      OUT     D7506.0  ; NST6_COMP_LIFTER_SELECT
; Rung 20
189   LDI     L1590  ; NST6 MAN OPERATION SEL BIT1
      AND     L1591  ; NST6 MAN OPERATION SEL BIT2
      ANI     L1592  ; NST6 MAN OPERATION SEL BIT4
      ANI     D7506.0  ; NST6_COMP_LIFTER_SELECT
      ANI     D7506.2  ; NST6_SEALING_UNIT_THREE_SELECT
      ANI     D7506.3  ; NST6_CHILD_ITEM_CHECK_SELECT
      ANI     D7506.4  ; NST6_MACHINE_PALLET_GATE_SELECT
      ANI     D7506.5  ; NST6_BUFFER_PALLET_GATE_SELECT
      OUT     D7506.1  ; NST6_SEALING_UNIT_1AND2_SELECT
; Rung 21
204   LD      L1590  ; NST6 MAN OPERATION SEL BIT1
      AND     L1591  ; NST6 MAN OPERATION SEL BIT2
      ANI     L1592  ; NST6 MAN OPERATION SEL BIT4
      ANI     D7506.0  ; NST6_COMP_LIFTER_SELECT
      ANI     D7506.1  ; NST6_SEALING_UNIT_1AND2_SELECT
      ANI     D7506.3  ; NST6_CHILD_ITEM_CHECK_SELECT
      ANI     D7506.4  ; NST6_MACHINE_PALLET_GATE_SELECT
      ANI     D7506.5  ; NST6_BUFFER_PALLET_GATE_SELECT
      OUT     D7506.2  ; NST6_SEALING_UNIT_THREE_SELECT
; Rung 22
219   LDI     L1590  ; NST6 MAN OPERATION SEL BIT1
      ANI     L1591  ; NST6 MAN OPERATION SEL BIT2
      AND     L1592  ; NST6 MAN OPERATION SEL BIT4
      ANI     D7506.0  ; NST6_COMP_LIFTER_SELECT
      ANI     D7506.1  ; NST6_SEALING_UNIT_1AND2_SELECT
      ANI     D7506.2  ; NST6_SEALING_UNIT_THREE_SELECT
      ANI     D7506.4  ; NST6_MACHINE_PALLET_GATE_SELECT
      ANI     D7506.5  ; NST6_BUFFER_PALLET_GATE_SELECT
      OUT     D7506.3  ; NST6_CHILD_ITEM_CHECK_SELECT
; Rung 23
234   LD      L1590  ; NST6 MAN OPERATION SEL BIT1
      ANI     L1591  ; NST6 MAN OPERATION SEL BIT2
      AND     L1592  ; NST6 MAN OPERATION SEL BIT4
      ANI     D7506.0  ; NST6_COMP_LIFTER_SELECT
      ANI     D7506.1  ; NST6_SEALING_UNIT_1AND2_SELECT
      ANI     D7506.2  ; NST6_SEALING_UNIT_THREE_SELECT
      ANI     D7506.3  ; NST6_CHILD_ITEM_CHECK_SELECT
      ANI     D7506.5  ; NST6_BUFFER_PALLET_GATE_SELECT
      OUT     D7506.4  ; NST6_MACHINE_PALLET_GATE_SELECT
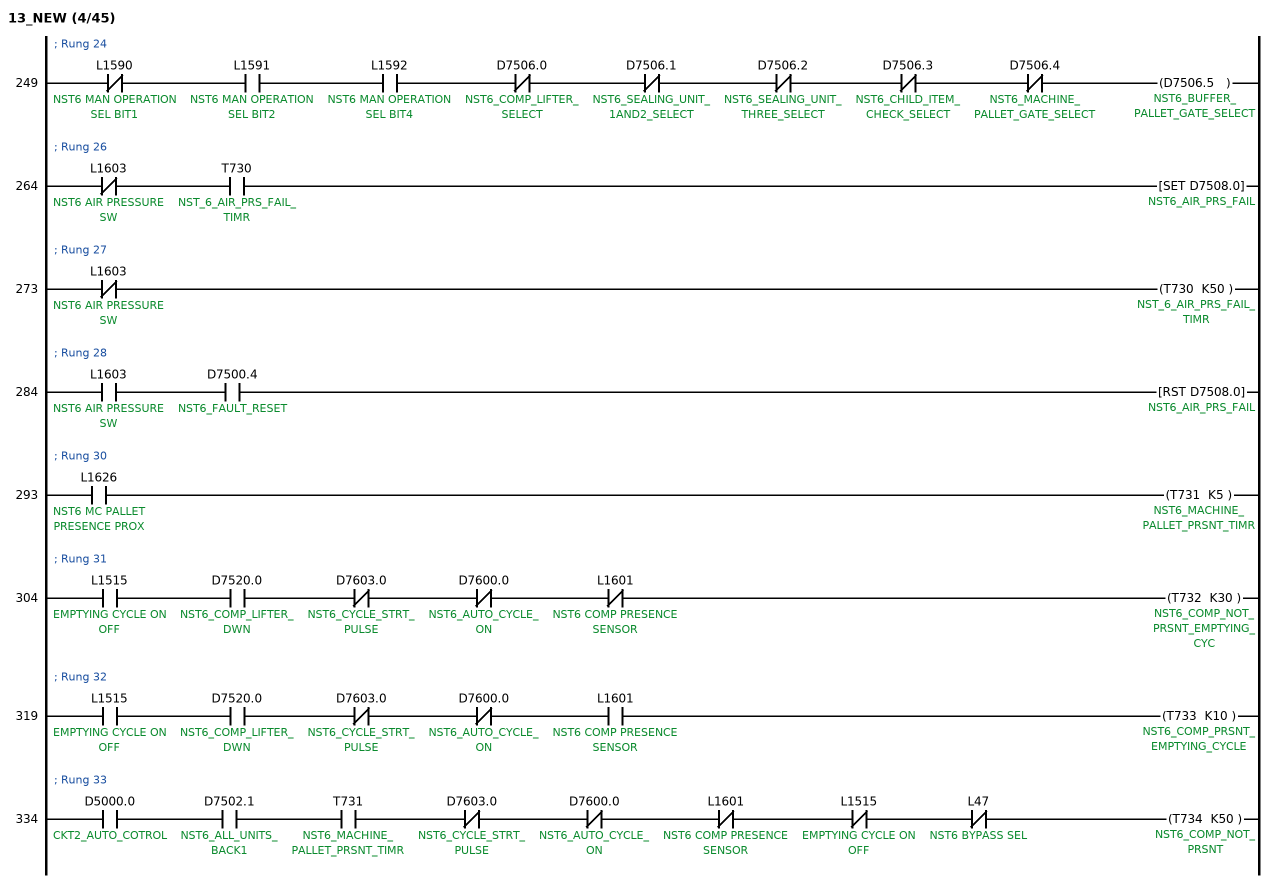
; Rung 24
249   LDI     L1590  ; NST6 MAN OPERATION SEL BIT1
      AND     L1591  ; NST6 MAN OPERATION SEL BIT2
      AND     L1592  ; NST6 MAN OPERATION SEL BIT4
      ANI     D7506.0  ; NST6_COMP_LIFTER_SELECT
      ANI     D7506.1  ; NST6_SEALING_UNIT_1AND2_SELECT
      ANI     D7506.2  ; NST6_SEALING_UNIT_THREE_SELECT
      ANI     D7506.3  ; NST6_CHILD_ITEM_CHECK_SELECT
      ANI     D7506.4  ; NST6_MACHINE_PALLET_GATE_SELECT
      OUT     D7506.5  ; NST6_BUFFER_PALLET_GATE_SELECT
; Rung 26
264   LDI     L1603  ; NST6 AIR PRESSURE SW
      AND     T730  ; NST_6_AIR_PRS_FAIL_TIMR
      SET     D7508.0  ; NST6_AIR_PRS_FAIL
; Rung 27
273   LDI     L1603  ; NST6 AIR PRESSURE SW
      OUT     T730 K50  ; NST_6_AIR_PRS_FAIL_TIMR
; Rung 28
284   LD      L1603  ; NST6 AIR PRESSURE SW
      AND     D7500.4  ; NST6_FAULT_RESET
      RST     D7508.0  ; NST6_AIR_PRS_FAIL
; Rung 30
293   LD      L1626  ; NST6 MC PALLET PRESENCE PROX
      OUT     T731 K5  ; NST6_MACHINE_PALLET_PRSNT_TIMR
; Rung 31
304   LD      L1515  ; EMPTYING CYCLE ON OFF
      AND     D7520.0  ; NST6_COMP_LIFTER_DWN
      ANI     D7603.0  ; NST6_CYCLE_STRT_PULSE
      ANI     D7600.0  ; NST6_AUTO_CYCLE_ON
      ANI     L1601  ; NST6 COMP PRESENCE SENSOR
      OUT     T732 K30  ; NST6_COMP_NOT_PRSNT_EMPTYING_CYC
; Rung 32
319   LD      L1515  ; EMPTYING CYCLE ON OFF
      AND     D7520.0  ; NST6_COMP_LIFTER_DWN
      ANI     D7603.0  ; NST6_CYCLE_STRT_PULSE
      ANI     D7600.0  ; NST6_AUTO_CYCLE_ON
      AND     L1601  ; NST6 COMP PRESENCE SENSOR
      OUT     T733 K10  ; NST6_COMP_PRSNT_EMPTYING_CYCLE
; Rung 33
334   LD      D5000.0  ; CKT2_AUTO_COTROL
      AND     D7502.1  ; NST6_ALL_UNITS_BACK1
      AND     T731  ; NST6_MACHINE_PALLET_PRSNT_TIMR
      ANI     D7603.0  ; NST6_CYCLE_STRT_PULSE
      ANI     D7600.0  ; NST6_AUTO_CYCLE_ON
      ANI     L1601  ; NST6 COMP PRESENCE SENSOR
      ANI     L1515  ; EMPTYING CYCLE ON OFF
      ANI     L47  ; NST6 BYPASS SEL
      OUT     T734 K50  ; NST6_COMP_NOT_PRSNT
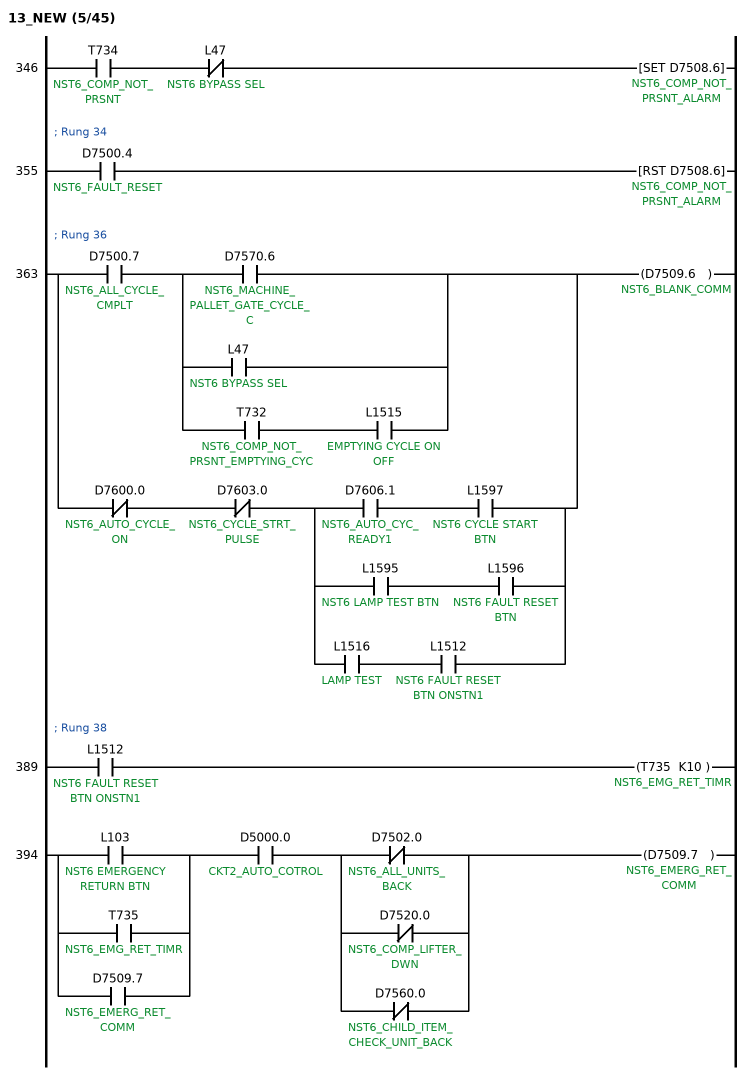
346   LD      T734  ; NST6_COMP_NOT_PRSNT
      ANI     L47  ; NST6 BYPASS SEL
      SET     D7508.6  ; NST6_COMP_NOT_PRSNT_ALARM
; Rung 34
355   LD      D7500.4  ; NST6_FAULT_RESET
      RST     D7508.6  ; NST6_COMP_NOT_PRSNT_ALARM
; Rung 36
363   LD      D7500.7  ; NST6_ALL_CYCLE_CMPLT
      LD      D7570.6  ; NST6_MACHINE_PALLET_GATE_CYCLE_C
      OR      L47  ; NST6 BYPASS SEL
      LD      T732  ; NST6_COMP_NOT_PRSNT_EMPTYING_CYC
      AND     L1515  ; EMPTYING CYCLE ON OFF
      ORB
      ANB
      LDI     D7600.0  ; NST6_AUTO_CYCLE_ON
      ANI     D7603.0  ; NST6_CYCLE_STRT_PULSE
      LD      D7606.1  ; NST6_AUTO_CYC_READY1
      AND     L1597  ; NST6 CYCLE START BTN
      LD      L1595  ; NST6 LAMP TEST BTN
      AND     L1596  ; NST6 FAULT RESET BTN
      ORB
      LD      L1516  ; LAMP TEST
      AND     L1512  ; NST6 FAULT RESET BTN ONSTN1
      ORB
      ANB
      ORB
      OUT     D7509.6  ; NST6_BLANK_COMM
; Rung 38
389   LD      L1512  ; NST6 FAULT RESET BTN ONSTN1
      OUT     T735 K10  ; NST6_EMG_RET_TIMR
394   LD      L103  ; NST6 EMERGENCY RETURN BTN
      OR      T735  ; NST6_EMG_RET_TIMR
      OR      D7509.7  ; NST6_EMERG_RET_COMM
      AND     D5000.0  ; CKT2_AUTO_COTROL
      LDI     D7502.0  ; NST6_ALL_UNITS_BACK
      ORI     D7520.0  ; NST6_COMP_LIFTER_DWN
      ORI     D7560.0  ; NST6_CHILD_ITEM_CHECK_UNIT_BACK
      ANB
      OUT     D7509.7  ; NST6_EMERG_RET_COMM
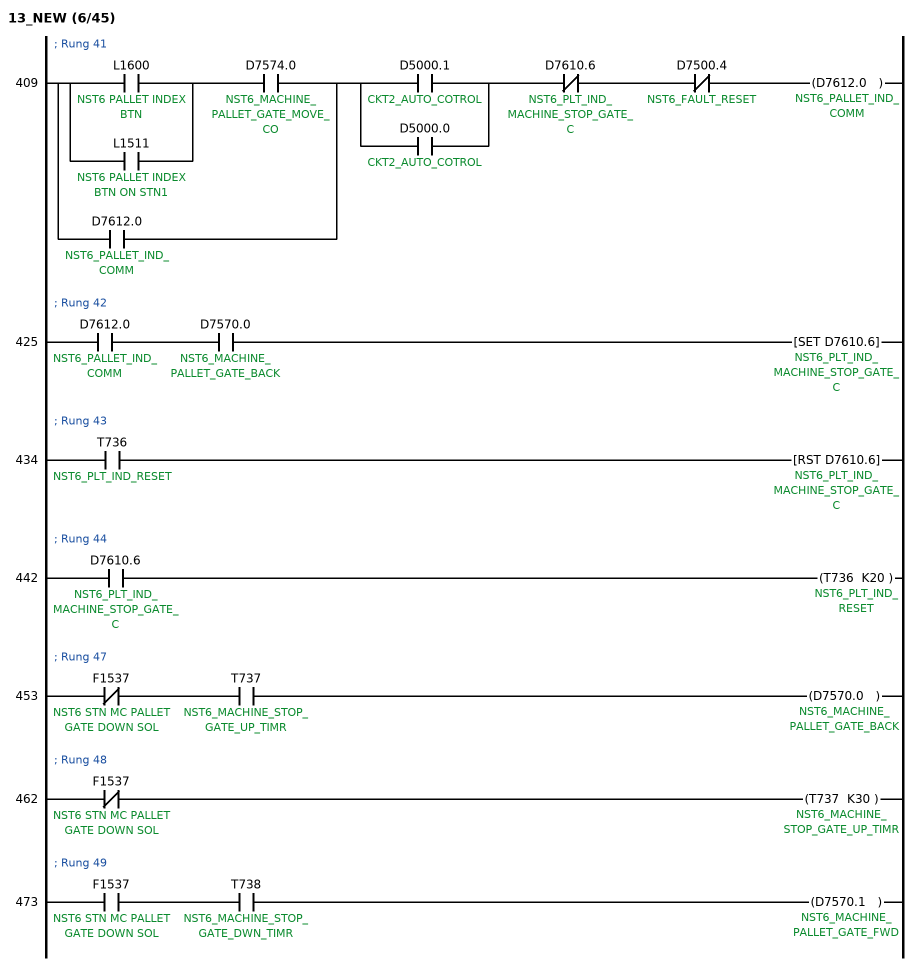
; Rung 41
409   LD      L1600  ; NST6 PALLET INDEX BTN
      OR      L1511  ; NST6 PALLET INDEX BTN ON STN1
      AND     D7574.0  ; NST6_MACHINE_PALLET_GATE_MOVE_CO
      OR      D7612.0  ; NST6_PALLET_IND_COMM
      LD      D5000.1  ; CKT2_AUTO_COTROL
      OR      D5000.0  ; CKT2_AUTO_COTROL
      ANB
      ANI     D7610.6  ; NST6_PLT_IND_MACHINE_STOP_GATE_C
      ANI     D7500.4  ; NST6_FAULT_RESET
      OUT     D7612.0  ; NST6_PALLET_IND_COMM
; Rung 42
425   LD      D7612.0  ; NST6_PALLET_IND_COMM
      AND     D7570.0  ; NST6_MACHINE_PALLET_GATE_BACK
      SET     D7610.6  ; NST6_PLT_IND_MACHINE_STOP_GATE_C
; Rung 43
434   LD      T736  ; NST6_PLT_IND_RESET
      RST     D7610.6  ; NST6_PLT_IND_MACHINE_STOP_GATE_C
; Rung 44
442   LD      D7610.6  ; NST6_PLT_IND_MACHINE_STOP_GATE_C
      OUT     T736 K20  ; NST6_PLT_IND_RESET
; Rung 47
453   LDI     F1537  ; NST6 STN MC PALLET GATE DOWN SOL
      AND     T737  ; NST6_MACHINE_STOP_GATE_UP_TIMR
      OUT     D7570.0  ; NST6_MACHINE_PALLET_GATE_BACK
; Rung 48
462   LDI     F1537  ; NST6 STN MC PALLET GATE DOWN SOL
      OUT     T737 K30  ; NST6_MACHINE_STOP_GATE_UP_TIMR
; Rung 49
473   LD      F1537  ; NST6 STN MC PALLET GATE DOWN SOL
      AND     T738  ; NST6_MACHINE_STOP_GATE_DWN_TIMR
      OUT     D7570.1  ; NST6_MACHINE_PALLET_GATE_FWD
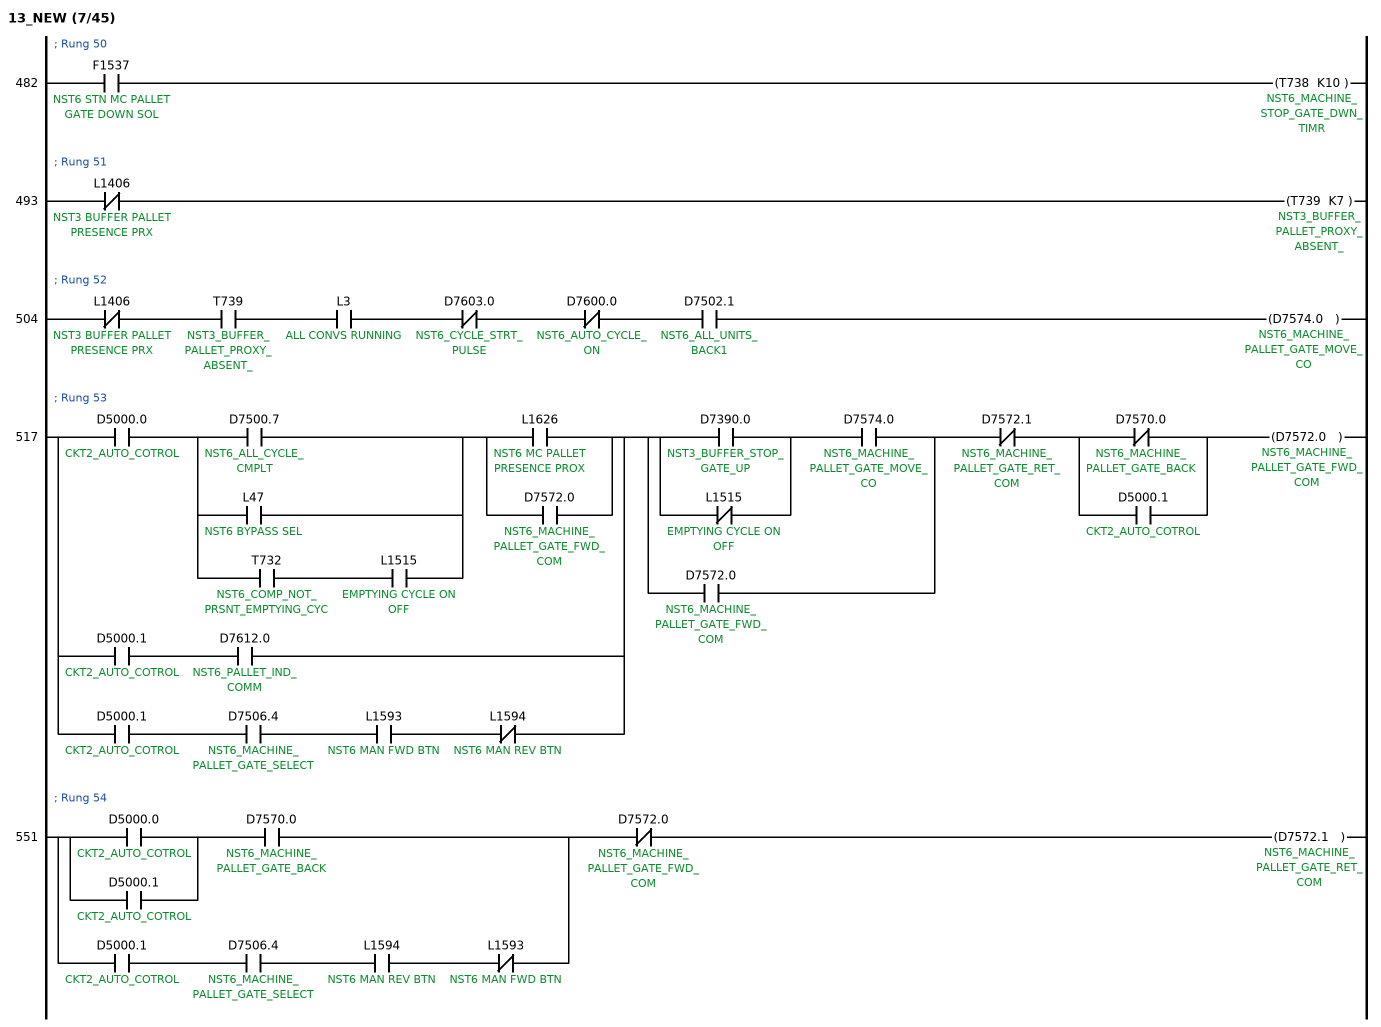
; Rung 50
482   LD      F1537  ; NST6 STN MC PALLET GATE DOWN SOL
      OUT     T738 K10  ; NST6_MACHINE_STOP_GATE_DWN_TIMR
; Rung 51
493   LDI     L1406  ; NST3 BUFFER PALLET PRESENCE PRX
      OUT     T739 K7  ; NST3_BUFFER_PALLET_PROXY_ABSENT_
; Rung 52
504   LDI     L1406  ; NST3 BUFFER PALLET PRESENCE PRX
      AND     T739  ; NST3_BUFFER_PALLET_PROXY_ABSENT_
      AND     L3  ; ALL CONVS RUNNING
      ANI     D7603.0  ; NST6_CYCLE_STRT_PULSE
      ANI     D7600.0  ; NST6_AUTO_CYCLE_ON
      AND     D7502.1  ; NST6_ALL_UNITS_BACK1
      OUT     D7574.0  ; NST6_MACHINE_PALLET_GATE_MOVE_CO
; Rung 53
517   LD      D5000.0  ; CKT2_AUTO_COTROL
      LD      D7500.7  ; NST6_ALL_CYCLE_CMPLT
      OR      L47  ; NST6 BYPASS SEL
      LD      T732  ; NST6_COMP_NOT_PRSNT_EMPTYING_CYC
      AND     L1515  ; EMPTYING CYCLE ON OFF
      ORB
      ANB
      LD      L1626  ; NST6 MC PALLET PRESENCE PROX
      OR      D7572.0  ; NST6_MACHINE_PALLET_GATE_FWD_COM
      ANB
      LD      D5000.1  ; CKT2_AUTO_COTROL
      AND     D7612.0  ; NST6_PALLET_IND_COMM
      ORB
      LD      D5000.1  ; CKT2_AUTO_COTROL
      AND     D7506.4  ; NST6_MACHINE_PALLET_GATE_SELECT
      AND     L1593  ; NST6 MAN FWD BTN
      ANI     L1594  ; NST6 MAN REV BTN
      ORB
      LD      D7390.0  ; NST3_BUFFER_STOP_GATE_UP
      ORI     L1515  ; EMPTYING CYCLE ON OFF
      AND     D7574.0  ; NST6_MACHINE_PALLET_GATE_MOVE_CO
      OR      D7572.0  ; NST6_MACHINE_PALLET_GATE_FWD_COM
      ANB
      ANI     D7572.1  ; NST6_MACHINE_PALLET_GATE_RET_COM
      LDI     D7570.0  ; NST6_MACHINE_PALLET_GATE_BACK
      OR      D5000.1  ; CKT2_AUTO_COTROL
      ANB
      OUT     D7572.0  ; NST6_MACHINE_PALLET_GATE_FWD_COM
; Rung 54
551   LD      D5000.0  ; CKT2_AUTO_COTROL
      OR      D5000.1  ; CKT2_AUTO_COTROL
      AND     D7570.0  ; NST6_MACHINE_PALLET_GATE_BACK
      LD      D5000.1  ; CKT2_AUTO_COTROL
      AND     D7506.4  ; NST6_MACHINE_PALLET_GATE_SELECT
      AND     L1594  ; NST6 MAN REV BTN
      ANI     L1593  ; NST6 MAN FWD BTN
      ORB
      ANI     D7572.0  ; NST6_MACHINE_PALLET_GATE_FWD_COM
      OUT     D7572.1  ; NST6_MACHINE_PALLET_GATE_RET_COM
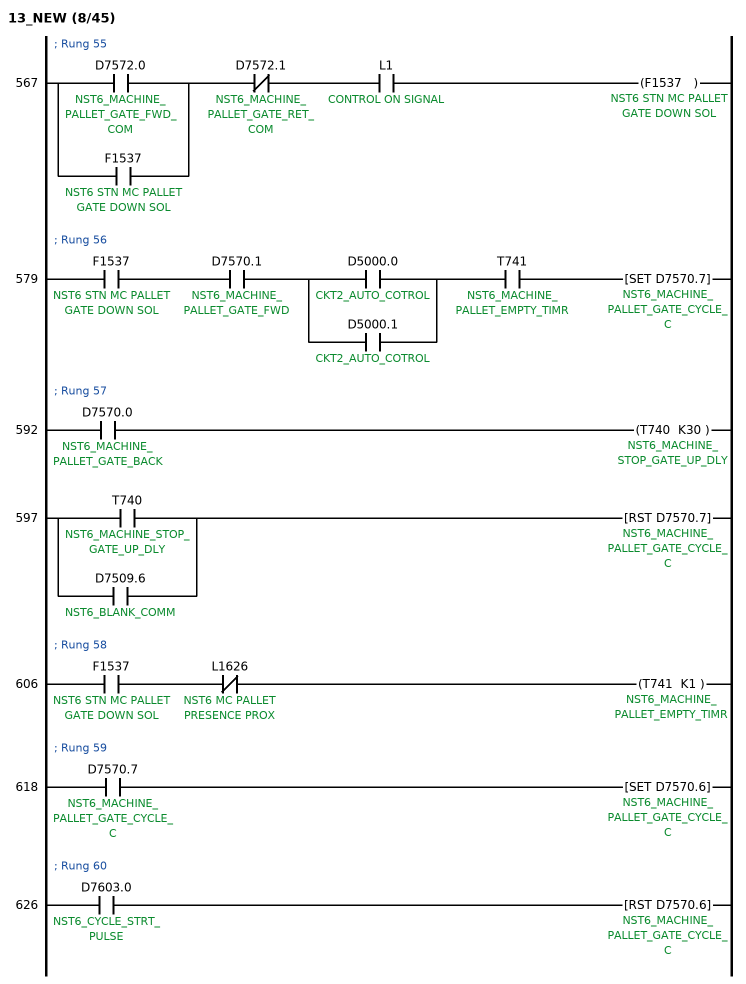
; Rung 55
567   LD      D7572.0  ; NST6_MACHINE_PALLET_GATE_FWD_COM
      OR      F1537  ; NST6 STN MC PALLET GATE DOWN SOL
      ANI     D7572.1  ; NST6_MACHINE_PALLET_GATE_RET_COM
      AND     L1  ; CONTROL ON SIGNAL
      OUT     F1537  ; NST6 STN MC PALLET GATE DOWN SOL
; Rung 56
579   LD      F1537  ; NST6 STN MC PALLET GATE DOWN SOL
      AND     D7570.1  ; NST6_MACHINE_PALLET_GATE_FWD
      LD      D5000.0  ; CKT2_AUTO_COTROL
      OR      D5000.1  ; CKT2_AUTO_COTROL
      ANB
      AND     T741  ; NST6_MACHINE_PALLET_EMPTY_TIMR
      SET     D7570.7  ; NST6_MACHINE_PALLET_GATE_CYCLE_C
; Rung 57
592   LD      D7570.0  ; NST6_MACHINE_PALLET_GATE_BACK
      OUT     T740 K30  ; NST6_MACHINE_STOP_GATE_UP_DLY
597   LD      T740  ; NST6_MACHINE_STOP_GATE_UP_DLY
      OR      D7509.6  ; NST6_BLANK_COMM
      RST     D7570.7  ; NST6_MACHINE_PALLET_GATE_CYCLE_C
; Rung 58
606   LD      F1537  ; NST6 STN MC PALLET GATE DOWN SOL
      ANI     L1626  ; NST6 MC PALLET PRESENCE PROX
      OUT     T741 K1  ; NST6_MACHINE_PALLET_EMPTY_TIMR
; Rung 59
618   LD      D7570.7  ; NST6_MACHINE_PALLET_GATE_CYCLE_C
      SET     D7570.6  ; NST6_MACHINE_PALLET_GATE_CYCLE_C
; Rung 60
626   LD      D7603.0  ; NST6_CYCLE_STRT_PULSE
      RST     D7570.6  ; NST6_MACHINE_PALLET_GATE_CYCLE_C
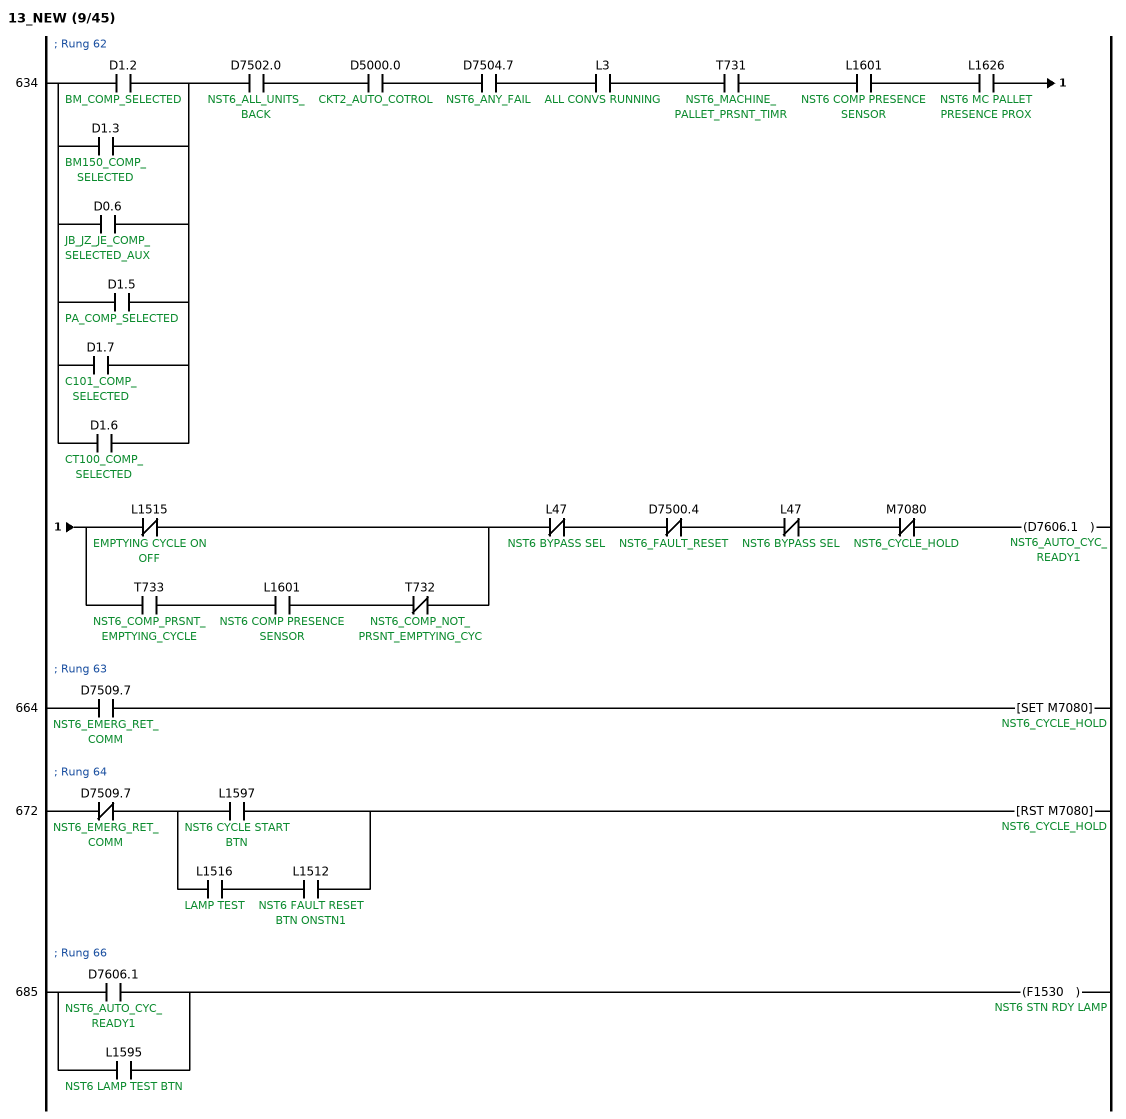
; Rung 62
634   LD      D1.2  ; BM_COMP_SELECTED
      OR      D1.3  ; BM150_COMP_SELECTED
      OR      D0.6  ; JB_JZ_JE_COMP_SELECTED_AUX
      OR      D1.5  ; PA_COMP_SELECTED
      OR      D1.7  ; C101_COMP_SELECTED
      OR      D1.6  ; CT100_COMP_SELECTED
      AND     D7502.0  ; NST6_ALL_UNITS_BACK
      AND     D5000.0  ; CKT2_AUTO_COTROL
      AND     D7504.7  ; NST6_ANY_FAIL
      AND     L3  ; ALL CONVS RUNNING
      AND     T731  ; NST6_MACHINE_PALLET_PRSNT_TIMR
      AND     L1601  ; NST6 COMP PRESENCE SENSOR
      AND     L1626  ; NST6 MC PALLET PRESENCE PROX
      LDI     L1515  ; EMPTYING CYCLE ON OFF
      LD      T733  ; NST6_COMP_PRSNT_EMPTYING_CYCLE
      AND     L1601  ; NST6 COMP PRESENCE SENSOR
      ANI     T732  ; NST6_COMP_NOT_PRSNT_EMPTYING_CYC
      ORB
      ANB
      ANI     L47  ; NST6 BYPASS SEL
      ANI     D7500.4  ; NST6_FAULT_RESET
      ANI     L47  ; NST6 BYPASS SEL
      ANI     M7080  ; NST6_CYCLE_HOLD
      OUT     D7606.1  ; NST6_AUTO_CYC_READY1
; Rung 63
664   LD      D7509.7  ; NST6_EMERG_RET_COMM
      SET     M7080  ; NST6_CYCLE_HOLD
; Rung 64
672   LDI     D7509.7  ; NST6_EMERG_RET_COMM
      LD      L1597  ; NST6 CYCLE START BTN
      LD      L1516  ; LAMP TEST
      AND     L1512  ; NST6 FAULT RESET BTN ONSTN1
      ORB
      ANB
      RST     M7080  ; NST6_CYCLE_HOLD
; Rung 66
685   LD      D7606.1  ; NST6_AUTO_CYC_READY1
      OR      L1595  ; NST6 LAMP TEST BTN
      OUT     F1530  ; NST6 STN RDY LAMP
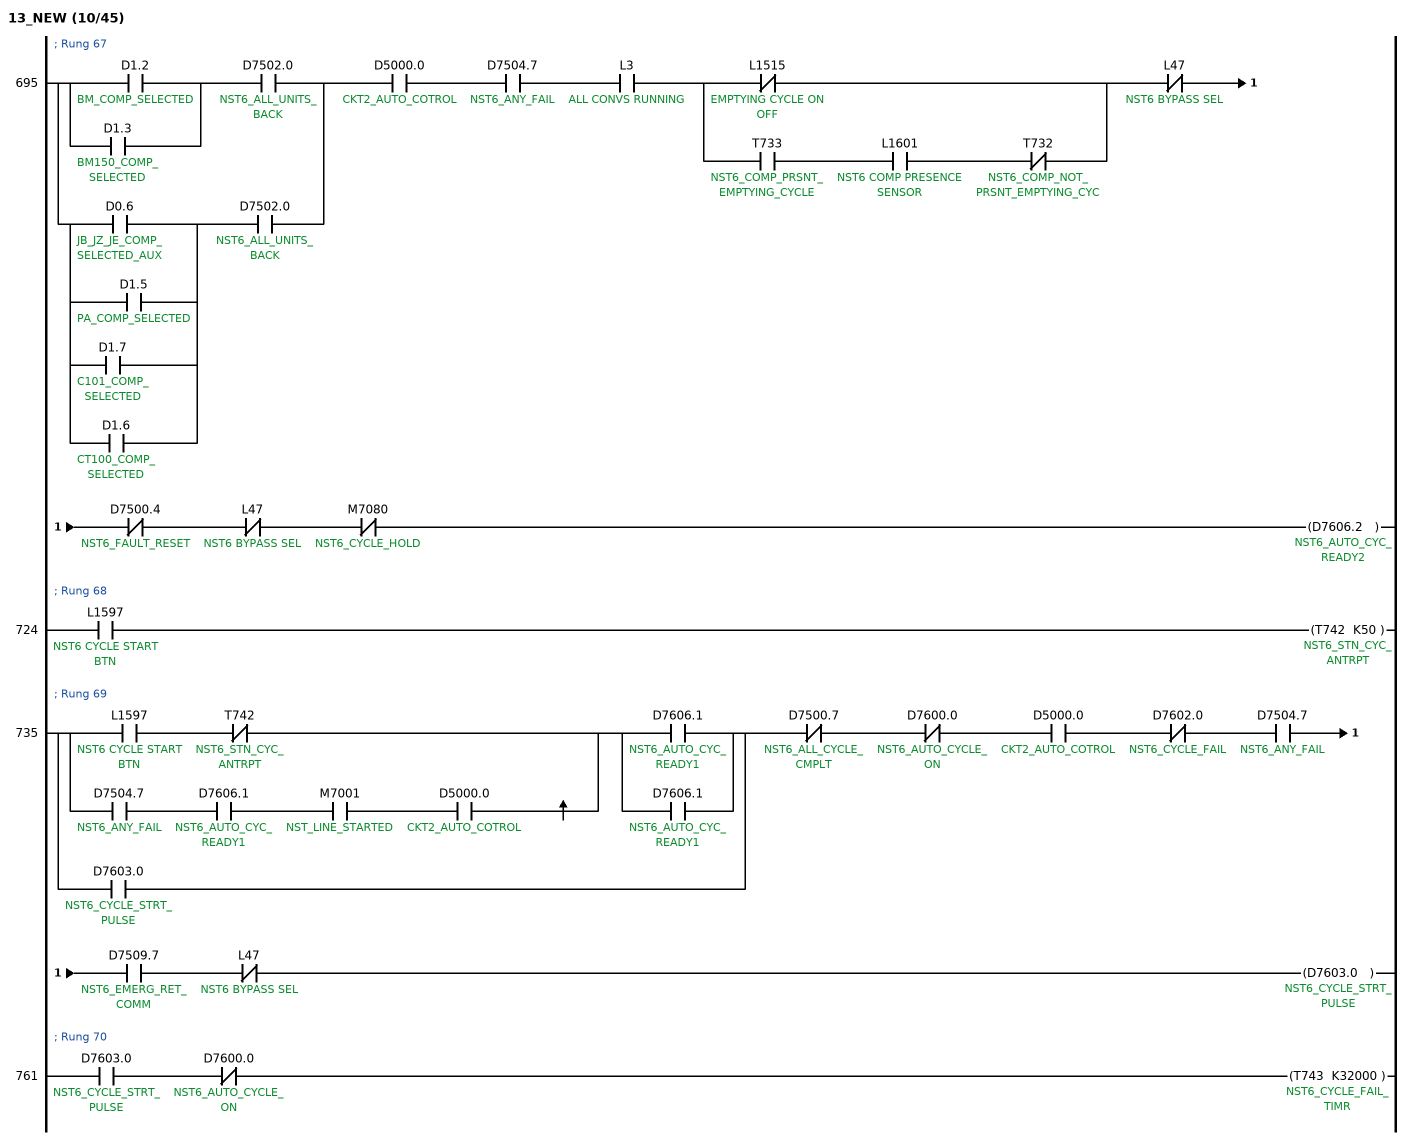
; Rung 67
695   LD      D1.2  ; BM_COMP_SELECTED
      OR      D1.3  ; BM150_COMP_SELECTED
      AND     D7502.0  ; NST6_ALL_UNITS_BACK
      LD      D0.6  ; JB_JZ_JE_COMP_SELECTED_AUX
      OR      D1.5  ; PA_COMP_SELECTED
      OR      D1.7  ; C101_COMP_SELECTED
      OR      D1.6  ; CT100_COMP_SELECTED
      AND     D7502.0  ; NST6_ALL_UNITS_BACK
      ORB
      AND     D5000.0  ; CKT2_AUTO_COTROL
      AND     D7504.7  ; NST6_ANY_FAIL
      AND     L3  ; ALL CONVS RUNNING
      LDI     L1515  ; EMPTYING CYCLE ON OFF
      LD      T733  ; NST6_COMP_PRSNT_EMPTYING_CYCLE
      AND     L1601  ; NST6 COMP PRESENCE SENSOR
      ANI     T732  ; NST6_COMP_NOT_PRSNT_EMPTYING_CYC
      ORB
      ANB
      ANI     L47  ; NST6 BYPASS SEL
      ANI     D7500.4  ; NST6_FAULT_RESET
      ANI     L47  ; NST6 BYPASS SEL
      ANI     M7080  ; NST6_CYCLE_HOLD
      OUT     D7606.2  ; NST6_AUTO_CYC_READY2
; Rung 68
724   LD      L1597  ; NST6 CYCLE START BTN
      OUT     T742 K50  ; NST6_STN_CYC_ANTRPT
; Rung 69
735   LD      L1597  ; NST6 CYCLE START BTN
      ANI     T742  ; NST6_STN_CYC_ANTRPT
      LD      D7504.7  ; NST6_ANY_FAIL
      AND     D7606.1  ; NST6_AUTO_CYC_READY1
      AND     M7001  ; NST_LINE_STARTED
      AND     D5000.0  ; CKT2_AUTO_COTROL
      MEP
      ORB
      LD      D7606.1  ; NST6_AUTO_CYC_READY1
      OR      D7606.1  ; NST6_AUTO_CYC_READY1
      ANB
      OR      D7603.0  ; NST6_CYCLE_STRT_PULSE
      ANI     D7500.7  ; NST6_ALL_CYCLE_CMPLT
      ANI     D7600.0  ; NST6_AUTO_CYCLE_ON
      AND     D5000.0  ; CKT2_AUTO_COTROL
      ANI     D7602.0  ; NST6_CYCLE_FAIL
      AND     D7504.7  ; NST6_ANY_FAIL
      AND     D7509.7  ; NST6_EMERG_RET_COMM
      ANI     L47  ; NST6 BYPASS SEL
      OUT     D7603.0  ; NST6_CYCLE_STRT_PULSE
; Rung 70
761   LD      D7603.0  ; NST6_CYCLE_STRT_PULSE
      ANI     D7600.0  ; NST6_AUTO_CYCLE_ON
      OUT     T743 K32000  ; NST6_CYCLE_FAIL_TIMR
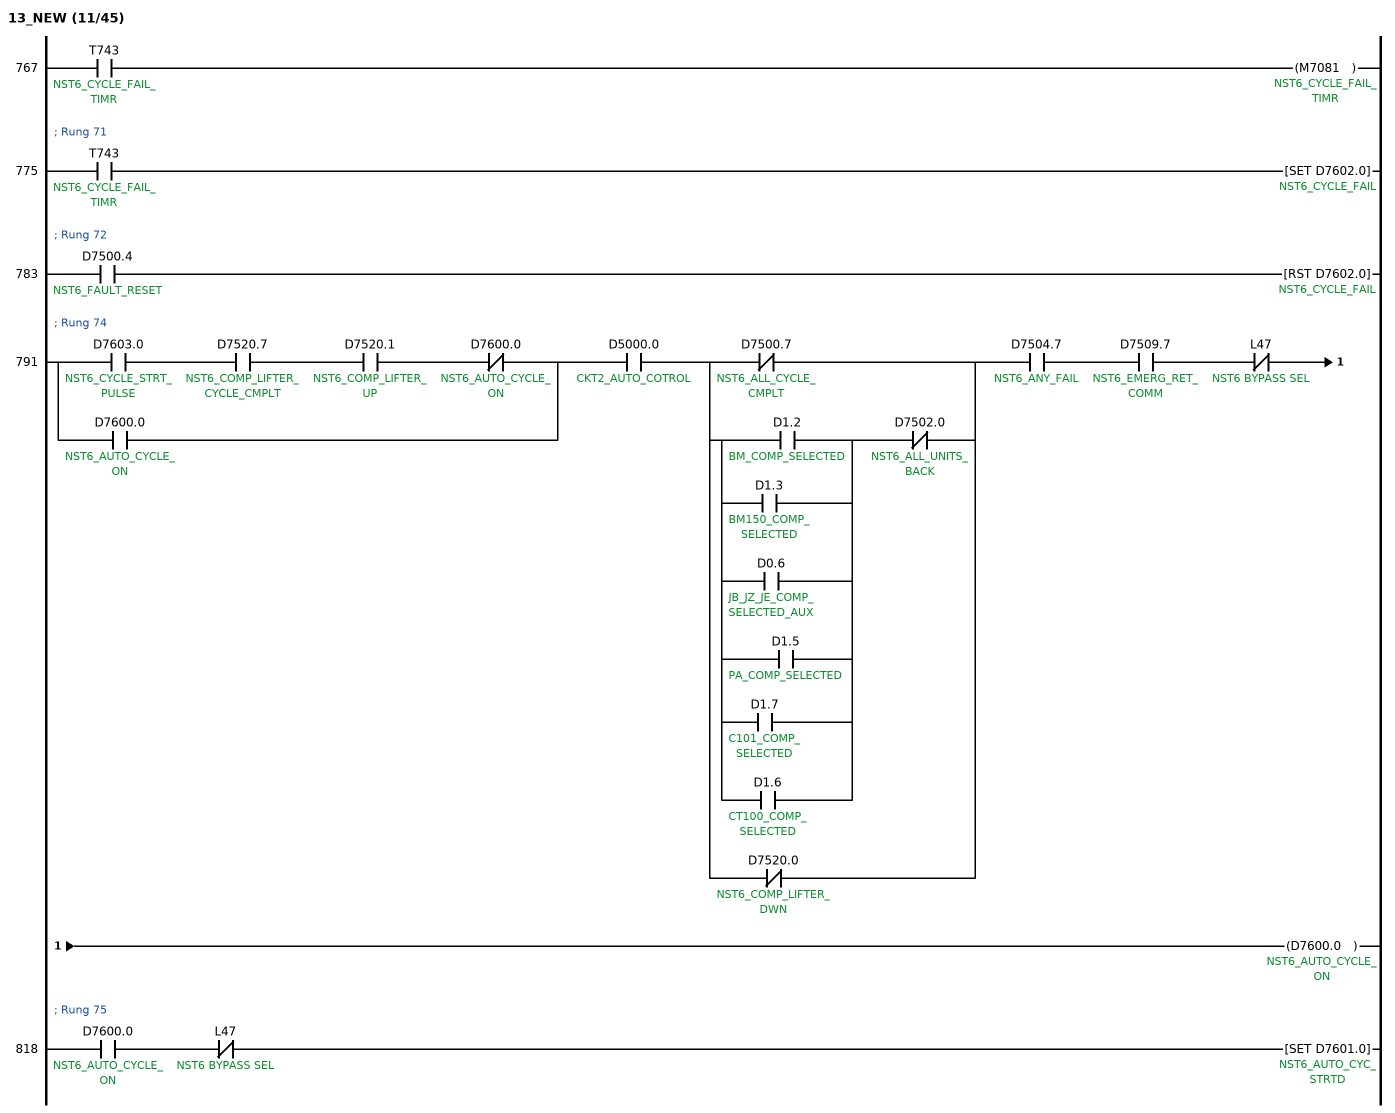
767   LD      T743  ; NST6_CYCLE_FAIL_TIMR
      OUT     M7081  ; NST6_CYCLE_FAIL_TIMR
; Rung 71
775   LD      T743  ; NST6_CYCLE_FAIL_TIMR
      SET     D7602.0  ; NST6_CYCLE_FAIL
; Rung 72
783   LD      D7500.4  ; NST6_FAULT_RESET
      RST     D7602.0  ; NST6_CYCLE_FAIL
; Rung 74
791   LD      D7603.0  ; NST6_CYCLE_STRT_PULSE
      AND     D7520.7  ; NST6_COMP_LIFTER_CYCLE_CMPLT
      AND     D7520.1  ; NST6_COMP_LIFTER_UP
      ANI     D7600.0  ; NST6_AUTO_CYCLE_ON
      OR      D7600.0  ; NST6_AUTO_CYCLE_ON
      AND     D5000.0  ; CKT2_AUTO_COTROL
      LDI     D7500.7  ; NST6_ALL_CYCLE_CMPLT
      LD      D1.2  ; BM_COMP_SELECTED
      OR      D1.3  ; BM150_COMP_SELECTED
      OR      D0.6  ; JB_JZ_JE_COMP_SELECTED_AUX
      OR      D1.5  ; PA_COMP_SELECTED
      OR      D1.7  ; C101_COMP_SELECTED
      OR      D1.6  ; CT100_COMP_SELECTED
      ANI     D7502.0  ; NST6_ALL_UNITS_BACK
      ORB
      ORI     D7520.0  ; NST6_COMP_LIFTER_DWN
      ANB
      AND     D7504.7  ; NST6_ANY_FAIL
      AND     D7509.7  ; NST6_EMERG_RET_COMM
      ANI     L47  ; NST6 BYPASS SEL
      OUT     D7600.0  ; NST6_AUTO_CYCLE_ON
; Rung 75
818   LD      D7600.0  ; NST6_AUTO_CYCLE_ON
      ANI     L47  ; NST6 BYPASS SEL
      SET     D7601.0  ; NST6_AUTO_CYC_STRTD
